// TIA Portal V17 program export: 9 tag tables, 18 data types, 15 data blocks, 39 code blocks (in call order from the OBs), 98 instance data blocks

VAR_GLOBAL   // PLC tag table "Check Scale Station-6"
   TAG_201 AT %M2.3 : Bool;
   TAG_202 AT %M2.4 : Bool;
   Tag_100 AT %M2.5 : Bool;
   "anti jammer_L2" AT %M2.6 : Bool;
   Tag_79_L2 AT %M2.7 : Bool;
   S5_STOPPER_SENSOR_l2 AT %M3.0 : Bool;
   S5_SENSOR_CYL7_DUMMY_TAG AT %M3.1 : Bool;
   Tag_102 AT %M3.2 : Bool;
   Seq_Lifttable_done_L2 AT %M3.3 : Bool;
   MC_Reset_L2 AT %M3.4 : Bool;
   TAG_203 AT %M3.5 : Bool;
   TAG_204 AT %M3.6 : Bool;
   TAG_205 AT %M3.7 : Bool;
   TAG_206 AT %M4.0 : Bool;
   TAG_207 AT %M4.1 : Bool;
   TAG_208 AT %M4.2 : Bool;
   TAG_209 AT %M4.3 : Bool;
   TAG210 AT %M4.4 : Bool;
   TAG211 AT %M4.5 : Bool;
   TAG216 AT %M4.6 : Bool;
   TAG213 AT %M4.7 : Bool;
   TAG214 AT %M5.0 : Bool;
   TAG215 AT %M5.1 : Bool;
   TAG217 AT %M5.2 : Bool;
   TAG218 AT %M5.3 : Bool;
   TAG212 AT %M5.4 : Bool;
   old_id AT %MW6 : Int;
   New_id AT %MW18 : Int;
END_VAR

VAR_GLOBAL   // PLC tag table "Common Tags"
END_VAR

VAR_GLOBAL   // PLC tag table "Correction Station-7"
END_VAR

VAR_GLOBAL   // PLC tag table "Default tag table"
   A_Tag_1 AT %M102.0 : Bool;
   A_Tag_2 AT %M102.1 : Bool;
   A_Tag_3 AT %M102.2 : Bool;
   A_Tag_4 AT %M102.3 : Bool;
   A_Tag_5 AT %M102.4 : Bool;
   Tag_1 AT %M200.0 : Bool;
   P_Trig08 AT %M2.0 : Bool;
   Tag_3 AT %M9.0 : Bool;
   Tag_4 AT %M9.1 : Bool;
   Tag_5 AT %M200.2 : Bool;
   A_Tag_11 AT %M2.1 : Bool;
   Tag_6 AT %M200.1 : Bool;
   Tag_7 AT %M110.0 : Bool;
   Tag_8 AT %M210.0 : Bool;
   Tag_9 AT %M210.1 : Bool;
   Tag_10 AT %M210.2 : Bool;
   Tag_11 AT %M210.4 : Bool;
   Tag_12 AT %M210.5 : Bool;
   Tag_13 AT %M210.6 : Bool;
   temp AT %M300.0 : Bool;
   Tag_14 AT %M210.7 : Bool;
   Tag_15 AT %M9.2 : Bool;
   Tag_17 AT %MW13 : Int;
   Tag_18 AT %MW15 : Int;
   Master1_Done_Bit AT %M11.0 : Bool;
   Master_Error_Bit AT %M11.1 : Bool;
   Tag_19 AT %MW500 : Word;
   Tag_20 AT %MW100 : Int;
   Tag_21 AT %M9.7 : Bool;
   Tag_22 AT %M20.0 : Bool;
   Tag_23 AT %M20.1 : Bool;
   Tag_24 AT %M22.0 : Bool;
   Tag_25 AT %M22.1 : Bool;
   System_Byte AT %MB1 : Byte;
   FirstScan AT %M1.0 : Bool;
   DiagStatusUpdate AT %M1.1 : Bool;
   AlwaysTRUE AT %M1.2 : Bool;
   AlwaysFALSE AT %M1.3 : Bool;
   Clock_Byte AT %MB0 : Byte;
   Clock_10Hz AT %M0.0 : Bool;
   Clock_5Hz AT %M0.1 : Bool;
   "Clock_2.5Hz" AT %M0.2 : Bool;
   Clock_2Hz AT %M0.3 : Bool;
   "Clock_1.25Hz" AT %M0.4 : Bool;
   Clock_1Hz AT %M0.5 : Bool;
   "Clock_0.625Hz" AT %M0.6 : Bool;
   "Clock_0.5Hz" AT %M0.7 : Bool;
   Tag_26 AT %M503.6 : Bool;
   Tag_27 AT %M23.0 : Bool;
   Tag_28 AT %M25.0 : Bool;
   Tag_29 AT %M25.1 : Bool;
   Tag_30 AT %M26.0 : Bool;
   Tag_31 AT %M27.0 : Bool;
   Tag_32 AT %M27.1 : Bool;
   Tag_33 AT %M27.2 : Bool;
   Tag_34 AT %M27.3 : Bool;
   Tag_35 AT %M27.4 : Bool;
   Tag_36 AT %M27.5 : Bool;
   Tag_37 AT %M27.6 : Bool;
   Tag_38 AT %M27.7 : Bool;
   Tag_39 AT %M28.0 : Bool;
   Tag_40 AT %M28.1 : Bool;
   Tag_41 AT %M28.2 : Bool;
   Tag_42 AT %M28.3 : Bool;
   Tag_43 AT %M28.4 : Bool;
   Tag_44 AT %M28.5 : Bool;
   Tag_45 AT %M28.6 : Bool;
   Tag_2 AT %M211.0 : Bool;
   Tag_16 AT %M211.2 : Bool;
   Tag_46 AT %M211.3 : Bool;
   Tag_47 AT %M212.0 : Bool;
   Tag_48 AT %M212.1 : Bool;
   Tag_49 AT %M212.2 : Bool;
   Tag_50 AT %M212.3 : Bool;
   Tag_51 AT %M212.4 : Bool;
   Tag_52 AT %M213.5 : Bool;
   Tag_53 AT %M212.5 : Bool;
   Tag_54 AT %M212.6 : Bool;
   Tag_55 AT %M212.7 : Bool;
   Tag_56 AT %M213.4 : Bool;
   Tag_57 AT %M213.0 : Bool;
   Tag_58 AT %M213.1 : Bool;
   Tag_59 AT %M213.2 : Bool;
   Tag_60 AT %M213.3 : Bool;
   Tag_61 AT %M214.0 : Bool;
   Tag_62 AT %M214.1 : Bool;
   Tag_63 AT %M214.2 : Bool;
   Tag_64 AT %M214.3 : Bool;
   Tag_65 AT %M214.4 : Bool;
   Tag_66 AT %M214.5 : Bool;
   Tag_67 AT %M214.6 : Bool;
   Tag_68 AT %MW1000 : Int;
   Tag_69 AT %M9.3 : Bool;
   Tag_70 AT %M214.7 : Bool;
   NUM_0 AT %I4.0 : Bool;
   NUM_1 AT %I4.1 : Bool;
   NUM_2 AT %I4.2 : Bool;
   NUM_3 AT %I4.3 : Bool;
   NUM_4 AT %I4.4 : Bool;
   NUM_5 AT %I4.5 : Bool;
   NUM_6 AT %I4.6 : Bool;
   NUM_7 AT %I4.7 : Bool;
   NUM_8 AT %I5.0 : Bool;
   NUM_9 AT %I5.1 : Bool;
   ENTER AT %I5.2 : Bool;
   Clear AT %I5.3 : Bool;
   Tag_71 AT %M2.2 : Bool;
   S5_SENSOR_CYL6 AT %I3.6 : Bool;
   S5_DOWN_CONVEYOR AT %I3.7 : Bool;
   SCREEN AT %I5.4 : Bool;
   BPCL_CY AT %I5.5 : Bool;
   MALABAR_GAS AT %I5.6 : Bool;
   "i5.7" AT %I5.7 : Bool;
   "q3.5" AT %Q3.5 : Bool;
   "q3.6" AT %Q3.6 : Bool;
   "q3.7" AT %Q3.7 : Bool;
   Tag_72 AT %M201.0 : Bool;
   Tag_73 AT %M201.1 : Bool;
   Tag_74 AT %M201.2 : Bool;
   Tag_75 AT %M99.7 : Bool;
   cylinder_pos AT %I2.4 : Bool;
   commercial AT %I2.5 : Bool;
   cylinder_exit AT %I2.6 : Bool;
   S5_CYCLE_START_L2 AT %I0.2 : Bool;
   S5_CYCLE_RESET_L2 AT %I0.3 : Bool;
   SEQ_RESET AT %I0.4 : Bool;
   MANUAL_SEQ AT %I0.5 : Bool;
   "i0.6" AT %I0.6 : Bool;
   "i0.7" AT %I0.7 : Bool;
   SEQ_RESET_L2 AT %I2.7 : Bool;
   S5_STOPPER_SENSOR AT %I3.0 : Bool;
   S5_SENSOR_CYL1 AT %I3.1 : Bool;
   S5_SENSOR_CYL2 AT %I3.2 : Bool;
   S5_SENSOR_CYL3 AT %I3.3 : Bool;
   S5_SENSOR_CYL4 AT %I3.4 : Bool;
   S5_SENSOR_CYL5 AT %I3.5 : Bool;
   DIVERTER AT %Q1.4 : Bool;
   PLC_LIVE AT %Q1.5 : Bool;
   spare_2 AT %Q1.6 : Bool;
   spare_3 AT %Q1.7 : Bool;
   S5_STOPPER_OP AT %Q2.0 : Bool;
   S5_LIFT_CYL6 AT %Q2.1 : Bool;
   S5_LIFT_CYL5 AT %Q2.2 : Bool;
   stopper AT %Q0.0 : Bool;
   Tag_76 AT %M888.7 : Bool;
   Tag_77 AT %M888.5 : Bool;
   Tag_78 AT %M888.6 : Bool;
   Seq_Lifttable_done AT %M100.7 : Bool;
   entry_data AT %MW90 : Int;
   MC_Reset AT %M100.2 : Bool;
   Tag_79 AT %M100.4 : Bool;
   "anti jammer" AT %M100.5 : Bool;
   Tag_80 AT %M100.6 : Bool;
   Tag_81 AT %M202.0 : Bool;
   Tag_82 AT %M202.1 : Bool;
   Tag_83 AT %M202.2 : Bool;
   Tag_84 AT %M202.4 : Bool;
   Tag_85 AT %M202.5 : Bool;
   Tag_86 AT %M202.6 : Bool;
   Tag_87 AT %M202.7 : Bool;
   Tag_88 AT %M203.0 : Bool;
   Tag_89 AT %M203.2 : Bool;
   Tag_90 AT %M203.1 : Bool;
   Tag_91 AT %M203.5 : Bool;
   Tag_92 AT %M203.7 : Bool;
   Tag_93 AT %M204.0 : Bool;
   Tag_94 AT %M204.1 : Bool;
   Tag_95 AT %M204.2 : Bool;
   Tag_96 AT %M204.3 : Bool;
   Tag_97 AT %M204.6 : Bool;
   Tag_98 AT %M203.4 : Bool;
   Tag_99 AT %M999.7 : Bool;
   Tag_101 AT %M5.7 : Bool;
   Tag_103 AT %M5.6 : Bool;
   Tag_104 AT %M500.0 : Bool;
   Tag_105 AT %M700.0 : Bool;
   Tag_106 AT %M700.1 : Bool;
   Check_Stopper AT %I6.0 : Bool;
   Check_presence AT %I6.1 : Bool;
   Check_pusher AT %I6.2 : Bool;
   Check_antijammer AT %I6.3 : Bool;
   Check_start_PB AT %I6.4 : Bool;
   Check_reset_PB AT %I6.5 : Bool;
   Check_Down_line_jammer AT %I6.6 : Bool;
   Correction_Stopper_sensor AT %I6.7 : Bool;
   Correction_Lift_sensor AT %I7.0 : Bool;
   Correction_Jammer_sensor AT %I7.1 : Bool;
   Correction_Start_PB AT %I7.2 : Bool;
   Correction_Reset_PB AT %I7.3 : Bool;
   Check_stopper_op AT %Q4.0 : Bool;
   Check_lift_table AT %Q4.1 : Bool;
   Check_pusher_op AT %Q4.2 : Bool;
   Correction_Stopper_solenoid AT %Q4.3 : Bool;
   Correction_Lift_solenoid AT %Q4.4 : Bool;
END_VAR

VAR_GLOBAL   // PLC tag table "Fine Filling Station-4"
   S4_CYCLE_START AT %I0.0 : Bool;
   S4_CYCLE_RESET AT %I0.1 : Bool;
   S4_STOPPER_SENSOR AT %I2.3 : Bool;
   S4_SENSOR_CYL1 AT %I1.1 : Bool;
   S4_SENSOR_CYL2 AT %I1.2 : Bool;
   S4_SENSOR_CYL3 AT %I1.3 : Bool;
   S4_SENSOR_CYL4 AT %I1.4 : Bool;
   S4_SENSOR_CYL5 AT %I1.5 : Bool;
   S4_SENSOR_CYL6 AT %I1.6 : Bool;
   SPARE_1 AT %I1.7 : Bool;
   MANUAL_SEQ_L2 AT %I2.0 : Bool;
   "i0.6_L2" AT %I2.1 : Bool;
   "i0.7_L2" AT %I2.2 : Bool;
   S4_DOWN_CONVEYOR AT %I1.0 : Bool;
   S4_STOPPER_OP AT %Q0.1 : Bool;
   S4_LIFT_CYL1 AT %Q0.2 : Bool;
   S4_LIFT_CYL2 AT %Q0.3 : Bool;
   S4_LIFT_CYL3 AT %Q0.4 : Bool;
   S4_LIFT_CYL4 AT %Q0.5 : Bool;
   S4_LIFT_CYL5 AT %Q0.6 : Bool;
   S4_LIFT_CYL6 AT %Q0.7 : Bool;
   S4_LIFT_CYL7 AT %Q1.0 : Bool;
   S4_LIFT_CYL8 AT %Q1.1 : Bool;
   S4_LIFT_CYL9 AT %Q1.2 : Bool;
   S4_LIFT_CYL10 AT %Q1.3 : Bool;
   S5_LIFT_CYL4 AT %Q2.3 : Bool;
   S5_LIFT_CYL3 AT %Q2.4 : Bool;
   S5_LIFT_CYL2 AT %Q2.5 : Bool;
   S5_LIFT_CYL1 AT %Q2.6 : Bool;
   spare_11 AT %Q2.7 : Bool;
   spare_12 AT %Q3.0 : Bool;
   spare_13 AT %Q3.1 : Bool;
   spare_14 AT %Q3.2 : Bool;
   spare_15 AT %Q3.3 : Bool;
   spare_16 AT %Q3.4 : Bool;
END_VAR

VAR_GLOBAL   // PLC tag table "Fine Filling Station-5"
END_VAR

VAR_GLOBAL   // PLC tag table "Pre Filling Station-2"
END_VAR

VAR_GLOBAL   // PLC tag table "Pre Filling Station-3"
END_VAR

VAR_GLOBAL   // PLC tag table "Tare Entry Station-1"
END_VAR

TYPE "Master_Step_No"
// stored: IsFailsafeCompliant false
   STRUCT
      Master_Step_No : Array[1..6] of USInt;
   END_STRUCT;
END_TYPE

TYPE "Mod_Client_Data"
// stored: IsFailsafeCompliant false
   STRUCT
      request : Bool;
      enable : Bool;
      disconnect : Bool;
      done : Bool;
      busy : Bool;
      error : Bool;
      status : Word;
      statusSave : Word;
      modbusMode : USInt;
      modbusDataAddress : UDInt;
      modbusDataLen : UInt;
   END_STRUCT;
END_TYPE

TYPE "Mod_Connect_Data"
// stored: IsFailsafeCompliant false
   STRUCT
      connectParamClient { S7_SetPoint := 'True'} : TCON_IP_v4;
   END_STRUCT;
   // connectParamClient.InterfaceId := 64;
   // connectParamClient.ID := 16#2;
   // connectParamClient.ActiveEstablished := true;
   // connectParamClient.RemoteAddress.ADDR[1] := 192;
   // connectParamClient.RemoteAddress.ADDR[2] := 168;
   // connectParamClient.RemoteAddress.ADDR[3] := 0;
   // connectParamClient.RemoteAddress.ADDR[4] := 3;
   // connectParamClient.RemotePort := 503;
   // connectParamClient.LocalPort := 0;
END_TYPE

TYPE "Mod_TCP_Data"
// stored: IsFailsafeCompliant false
   STRUCT
      Mod_TCP_Connect : "Mod_Connect_Data";
      Mod_Client { S7_SetPoint := 'True'} : Array[1..6] of "Mod_Client_Data";
   END_STRUCT;
END_TYPE

TYPE "uCylinderData"
// stored: IsFailsafeCompliant false
   STRUCT
      rCylinderID : Int;
      rNet_weight : Real;
      rTareWeight : Real;
      rGross_Weight : Real;
      iCylinderType : Int;   // 0=Domestic Cylinder; 1= Commercial
      iResult : Int;
   END_STRUCT;
END_TYPE

TYPE "ufinefill_station"
// stored: IsFailsafeCompliant false
   STRUCT
      INxNear_Filter_Stopper_L1 : Bool;
      INxFilling_Unit_L2 : Bool;
      INxFilling_Unit_L3 : Bool;
      INxFilling_Unit_L4 : Bool;
      INxFilling_Unit_L5 : Bool;
      INxDown_Line_Conveyor_L6 : Bool;
      INxCylinder_Selection_2 : Bool;
      INxCylinder_Selection_3 : Bool;
      INxCylinder_Selection_4 : Bool;
      INxStopper_Bypass_L2 : Bool;
      INxStopper_Bypass_L3 : Bool;
      INxStopper_Bypass_L4 : Bool;
      OUTxSolenoid_Control_Stopper_L1 : Bool;
      OUTxSolenoid_Control_LiftTable_L2 : Bool;
      OUTxSolenoid_Control_LiftTable_L3 : Bool;
      OUTxSolenoid_Control_LiftTable_L4 : Bool;
      OUTxSolenoid_Control_LiftTable_L5 : Bool;
      iSensingTime : Time;
      OUTxCylinder_Indicator_2 : Bool;
      OUTxCylinder_Indicator_3 : Bool;
      OUTxCylinder_Indicator_4 : Bool;
   END_STRUCT;
END_TYPE

TYPE "ufinefillingstation_general"
// stored: IsFailsafeCompliant false
   STRUCT
      INxCycle_Start : Bool;
      INxCycle_Reset : Bool;
   END_STRUCT;
END_TYPE

TYPE "LPG_CHECK_DATA"
// stored: IsFailsafeCompliant false
   STRUCT
      CHECK_SEQ_IN : Struct
         Cyl_IN_Pos : Bool;
         Auto_Start_Seq : Bool;
         Man_Start_Seq : Bool;
         Stop_Seq : Bool;
         Start_Timeout_Sec : DInt;
         Reset_Seq : Bool;
         Cylinder_Type : Int;
         Tare_Entry_SP : Real;
      END_STRUCT;
      CHECK_SEQ_OUT : Struct
         Checked_Status : Array[1..3] of Bool;
         Domestic_Cyl : Bool;
         Commercial_Cyl : Bool;
         Start_Timeout : Bool;
         Tare_Entry_Error : Bool;
         Filling_Error : Bool;
         Step_No : Int;
         Modbus_Busy : Bool;
      END_STRUCT;
   END_STRUCT;
END_TYPE

TYPE "LPG_FILL_DATA"
// stored: IsFailsafeCompliant false
   STRUCT
      FILL_SEQ_IN : Struct
         Cyl_IN_Pos : Bool;
         Auto_Start_Seq : Bool;
         Man_Start_Seq : Bool;
         Stop_Seq : Bool;
         Start_Timeout_Sec : DInt;
         Reset_Seq : Bool;
         Cylinder_Type : Int;
         Tare_Entry_SP : Real;
      END_STRUCT;
      FILL_SEQ_OUT : Struct
         Filled_Dat : Array[1..3] of Real;
         Domestic_Cyl : Bool;
         Commercial_Cyl : Bool;
         Start_Timeout : Bool;
         Tare_Entry_Error : Bool;
         Filling_Error : Bool;
         Step_No : Int;
         Modbus_Busy : Bool;
      END_STRUCT;
   END_STRUCT;
END_TYPE

TYPE "LPG_FILL_DATA_1"
// stored: IsFailsafeCompliant false
   STRUCT
      FILL_SEQ_IN : Struct
         Cyl_IN_Pos : Bool;
         Auto_Start_Seq : Bool;
         Man_Start_Seq : Bool;
         Stop_Seq : Bool;
         Start_Timeout_Sec : DInt;
         Reset_Seq : Bool;
         Cylinder_Type : Int;
         Tare_Entry_SP : Real;
      END_STRUCT;
      FILL_SEQ_OUT : Struct
         Filled_Dat : Array[1..10] of Real;
         Domestic_Cyl : Bool;
         Commercial_Cyl : Bool;
         Start_Timeout : Bool;
         Tare_Entry_Error : Bool;
         Filling_Error : Bool;
         Step_No : Int;
         Modbus_Busy : Bool;
      END_STRUCT;
   END_STRUCT;
END_TYPE

TYPE "MASTER_STATION"
// stored: IsFailsafeCompliant false
   STRUCT
      MODBUS_MASTER : Array[1..6] of "MOD_MASTER";
   END_STRUCT;
END_TYPE

TYPE "MODBUS_READ"
// stored: IsFailsafeCompliant false
   STRUCT
      MOD_COIL_DATA : Array[1..32] of Bool;
      MOD_HOLD_DATA_1 : Array[1..6] of Word;
      MOD_HOLD_DATA_2 : Array[1..2] of Word;
   END_STRUCT;
   // // MOD_COIL_DATA[1] : Satble Flag
   // // MOD_COIL_DATA[2] : Net Gross Flag
   // // MOD_COIL_DATA[3] : Operating Mode
   // // MOD_COIL_DATA[4] : Start Key Status
   // // MOD_COIL_DATA[5] : Zero Key Status
   // // MOD_COIL_DATA[6] : Tare Key Status
   // // MOD_COIL_DATA[7] : Print Key Status
   // // MOD_COIL_DATA[8] : Power On Zero
   // // MOD_COIL_DATA[9] : One Touch Zero Calibration
   // // MOD_COIL_DATA[10] : Under Weight Flag
   // // MOD_COIL_DATA[11] : Over Weight Flag
   // // MOD_COIL_DATA[12] : Gross Sign
   // // MOD_COIL_DATA[13] : Net Sign
   // // MOD_COIL_DATA[14] : Filled or Checked Data Status(W)
   // // MOD_COIL_DATA[15] : NA
   // // MOD_COIL_DATA[16] : Gate Input
   // // MOD_COIL_DATA[17] : Coarse Output
   // // MOD_COIL_DATA[18] : Fine Output
   // // MOD_COIL_DATA[19] : Batch Over Output
   // // MOD_COIL_DATA[20] : Gate Output
   // // MOD_COIL_DATA[21] : Lifter Output
   // // MOD_COIL_DATA[22] : Jam Output
   // // MOD_COIL_DATA[23] : NA
   // // MOD_COIL_DATA[24] : Indicator is in Parameter / Tare Entry Settings
   // // MOD_COIL_DATA[25] : Filling ON Status
   // // MOD_COIL_DATA[26] : Filling Time Over (W)
   // // MOD_COIL_DATA[27] : Tare Request Status
   // // MOD_COIL_DATA[28] : Filling Over Status
   // // MOD_COIL_DATA[29] : Filling Error Status(W)
   // // MOD_COIL_DATA[30] : Stop Filling (W)
   // // MOD_COIL_DATA[31] : Start Filling (W)
   // // MOD_COIL_DATA[32] : Tare Entry Error
   // // MOD_HOLD_DATA_1[2] : Fiiled Gross Weight
   // // MOD_HOLD_DATA_1[4] : Filled Net Weight
   // // MOD_HOLD_DATA_1[6] : Punched Tare Weight
   // // MOD_HOLD_DATA_2[2] : Fiiled Gross Weight
END_TYPE

TYPE "MODBUS_READ_1"
// stored: IsFailsafeCompliant false
   STRUCT
      MOD_COIL_DATA : Array[1..32] of Bool;
      MOD_HOLD_DATA_1 : Array[1..10] of Word;
      MOD_HOLD_DATA_2 : Array[1..2] of Word;
   END_STRUCT;
   // // MOD_COIL_DATA[1] : Satble Flag
   // // MOD_COIL_DATA[2] : Net Gross Flag
   // // MOD_COIL_DATA[3] : Operating Mode
   // // MOD_COIL_DATA[4] : Start Key Status
   // // MOD_COIL_DATA[5] : Zero Key Status
   // // MOD_COIL_DATA[6] : Tare Key Status
   // // MOD_COIL_DATA[7] : Print Key Status
   // // MOD_COIL_DATA[8] : Power On Zero
   // // MOD_COIL_DATA[9] : One Touch Zero Calibration
   // // MOD_COIL_DATA[10] : Under Weight Flag
   // // MOD_COIL_DATA[11] : Over Weight Flag
   // // MOD_COIL_DATA[12] : Gross Sign
   // // MOD_COIL_DATA[13] : Net Sign
   // // MOD_COIL_DATA[14] : Filled or Checked Data Status(W)
   // // MOD_COIL_DATA[15] : NA
   // // MOD_COIL_DATA[16] : Gate Input
   // // MOD_COIL_DATA[17] : Coarse Output
   // // MOD_COIL_DATA[18] : Fine Output
   // // MOD_COIL_DATA[19] : Batch Over Output
   // // MOD_COIL_DATA[20] : Gate Output
   // // MOD_COIL_DATA[21] : Lifter Output
   // // MOD_COIL_DATA[22] : Jam Output
   // // MOD_COIL_DATA[23] : NA
   // // MOD_COIL_DATA[24] : Indicator is in Parameter / Tare Entry Settings
   // // MOD_COIL_DATA[25] : Filling ON Status
   // // MOD_COIL_DATA[26] : Filling Time Over (W)
   // // MOD_COIL_DATA[27] : Tare Request Status
   // // MOD_COIL_DATA[28] : Filling Over Status
   // // MOD_COIL_DATA[29] : Filling Error Status(W)
   // // MOD_COIL_DATA[30] : Stop Filling (W)
   // // MOD_COIL_DATA[31] : Start Filling (W)
   // // MOD_COIL_DATA[32] : Tare Entry Error
   // // MOD_HOLD_DATA_1[2] : Fiiled Gross Weight
   // // MOD_HOLD_DATA_1[4] : Filled Net Weight
   // // MOD_HOLD_DATA_1[6] : Punched Tare Weight
   // // MOD_HOLD_DATA_2[2] : Fiiled Gross Weight
END_TYPE

TYPE "MODBUS_WRITE"
// stored: IsFailsafeCompliant false
   STRUCT
      MOD_COIL_DATA : Array[1..32] of Bool;
      MOD_HOLD_DATA_1 : Array[1..2] of Word;
      MOD_HOLD_DATA_2 : Array[1..2] of Word;
   END_STRUCT;
   // // MOD_COIL_DATA[1] : Satble Flag
   // // MOD_COIL_DATA[2] : Net Gross Flag
   // // MOD_COIL_DATA[3] : Operating Mode
   // // MOD_COIL_DATA[4] : Start Key Status
   // // MOD_COIL_DATA[5] : Zero Key Status
   // // MOD_COIL_DATA[6] : Tare Key Status
   // // MOD_COIL_DATA[7] : Print Key Status
   // // MOD_COIL_DATA[8] : Power On Zero
   // // MOD_COIL_DATA[9] : One Touch Zero Calibration
   // // MOD_COIL_DATA[10] : Under Weight Flag
   // // MOD_COIL_DATA[11] : Over Weight Flag
   // // MOD_COIL_DATA[12] : Gross Sign
   // // MOD_COIL_DATA[13] : Net Sign
   // // MOD_COIL_DATA[14] : Filled or Checked Data Status(W)
   // // MOD_COIL_DATA[15] : NA
   // // MOD_COIL_DATA[16] : Gate Input
   // // MOD_COIL_DATA[17] : Coarse Output
   // // MOD_COIL_DATA[18] : Fine Output
   // // MOD_COIL_DATA[19] : Batch Over Output
   // // MOD_COIL_DATA[20] : Gate Output
   // // MOD_COIL_DATA[21] : Lifter Output
   // // MOD_COIL_DATA[22] : Jam Output
   // // MOD_COIL_DATA[23] : NA
   // // MOD_COIL_DATA[24] : Indicator is in Parameter / Tare Entry Settings
   // // MOD_COIL_DATA[25] : Filling ON Status
   // // MOD_COIL_DATA[26] : Filling Time Over (W)
   // // MOD_COIL_DATA[27] : Tare Request Status
   // // MOD_COIL_DATA[28] : Filling Over Status
   // // MOD_COIL_DATA[29] : Filling Error Status(W)
   // // MOD_COIL_DATA[30] : Stop Filling (W)
   // // MOD_COIL_DATA[31] : Start Filling (W)
   // // MOD_COIL_DATA[32] : Tare Entry Error
   // // MOD_HOLD_DATA_1[2] : Cylinder Tare Weight
   // // MOD_HOLD_DATA_2[2] : Cylinder Tare Weight
END_TYPE

TYPE "MOD_COMM_LOAD"
// stored: IsFailsafeCompliant false
   STRUCT
      BAUD : UDInt;
      PARITY : UInt;
      FLOW_CTRL : UInt;
      RTS_ON_DLY : UInt;
      RTS_OFF_DLY : UInt;
      RESP_TO : UInt;
      DONE : Bool;
      ERROR : Bool;
      STATUS : Word;
   END_STRUCT;
END_TYPE

TYPE "MOD_MASTER"
// stored: IsFailsafeCompliant false
   STRUCT
      REQ : Bool;
      ADDR : UInt;
      MODE : USInt;
      DATA_ADDR : UDInt;
      DATA_LEN : UInt;
      DONE : Bool;
      BUSY : Bool;
      ERROR : Bool;
      STATUS : Word;
   END_STRUCT;
END_TYPE

TYPE "MOD_MASTER_DATA"
// stored: IsFailsafeCompliant false
   STRUCT
      MASTER_READ_DATA { S7_SetPoint := 'True'} : "MODBUS_READ";
      MASTER_WRITE_DATA { S7_SetPoint := 'True'} : "MODBUS_WRITE";
   END_STRUCT;
END_TYPE

TYPE "MOD_MASTER_DATA_1"
// stored: IsFailsafeCompliant false
   STRUCT
      MASTER_READ_DATA { S7_SetPoint := 'True'} : "MODBUS_READ_1";
      MASTER_WRITE_DATA { S7_SetPoint := 'True'} : "MODBUS_WRITE";
   END_STRUCT;
END_TYPE

DATA_BLOCK "Check_scale_Report"   // DB2001
{ S7_Optimized_Access := 'TRUE' }
VERSION : 0.1
// stored: AutoNumber false, DBAccessibleFromOPCUA true, IsOnlyStoredInLoadMemory false, IsRetainMemResEnabled false, IsWriteProtectedInAS false, MemoryReserve 100
   VAR
      Check_SCALE_DATA : "uCylinderData";
      Check_SCALE_DONE { S7_SetPoint := 'True'} : Bool;
   END_VAR
BEGIN
END_DATA_BLOCK

DATA_BLOCK "MASTER_FILL_DATA"   // DB105
{ S7_Optimized_Access := 'FALSE' }
VERSION : 0.1
// stored: AutoNumber false, DBAccessibleFromOPCUA true, IsOnlyStoredInLoadMemory false, IsWriteProtectedInAS false
   VAR
      FILL_STATION_4 : Array[1..6] of "LPG_FILL_DATA";
      FILL_STATION_5 : Array[1..6] of "LPG_FILL_DATA";
      CHECK_SCALE_1 { S7_SetPoint := 'True'} : "LPG_FILL_DATA_1";
      CORRECTION_SCALE { S7_SetPoint := 'True'} : "LPG_FILL_DATA";
   END_VAR
BEGIN
END_DATA_BLOCK

DATA_BLOCK "MASTER_SETUP_DB"   // DB13
{ S7_Optimized_Access := 'FALSE' }
VERSION : 0.1
// stored: AutoNumber true, DBAccessibleFromOPCUA true, IsOnlyStoredInLoadMemory false, IsWriteProtectedInAS false
   VAR RETAIN
      Enable_Station1 : Bool;
      Enable_Station4 : Bool;
      S1_Enabled_Station : Array[1..6] of Bool;
      S4_Enabled_Station : Array[1..6] of Bool;
      S1_Total_Station : Int;
      S4_Total_Station : Int;
      Enabled_Station_S1 : Int;
      Enabled_Station_S4 : Int;
      Enabled_Station_S5 : Int;
      S5_Enabled_Station : Array[1..6] of Bool;
      S5_Total_Station : Int;
      Enable_Station5 : Bool;
   END_VAR
BEGIN
END_DATA_BLOCK

DATA_BLOCK "MASTER_TCP_DATA"   // DB104
{ S7_Optimized_Access := 'FALSE' }
VERSION : 0.1
// stored: AutoNumber false, DBAccessibleFromOPCUA true, IsOnlyStoredInLoadMemory false, IsWriteProtectedInAS false
   VAR
      MOD_DEVICE_STATION4 : Array[1..6] of "MOD_MASTER_DATA";
      MOD_DEVICE_STATION5 : Array[1..6] of "MOD_MASTER_DATA";
      CHECK_SCALE_1 { S7_SetPoint := 'True'} : "MOD_MASTER_DATA_1";
      CORRECTION_SCALE { S7_SetPoint := 'True'} : "MOD_MASTER_DATA_1";
   END_VAR
BEGIN
END_DATA_BLOCK

DATA_BLOCK "MODBUS_DATA_READ"   // DB101
{ S7_Optimized_Access := 'FALSE' }
VERSION : 0.1
// stored: AutoNumber false, DBAccessibleFromOPCUA true, IsOnlyStoredInLoadMemory false, IsWriteProtectedInAS false
   VAR
      MOD_RD_DEV_STN4 : Array[1..6] of "MODBUS_READ";
      MOD_RD_DEV_STN5 : Array[1..6] of "MODBUS_READ";
      MOD_RD_DEV_CHECK_SCALE { S7_SetPoint := 'True'} : "MODBUS_READ_1";
      MOD_RD_DEV_CORRECTION_SCALE { S7_SetPoint := 'True'} : "MODBUS_READ_1";
   END_VAR
BEGIN
END_DATA_BLOCK

DATA_BLOCK "MODBUS_DATA_WRITE"   // DB102
{ S7_Optimized_Access := 'FALSE' }
VERSION : 0.1
// stored: AutoNumber false, DBAccessibleFromOPCUA true, IsOnlyStoredInLoadMemory false, IsWriteProtectedInAS false
   VAR
      MOD_WR_DEV_STN4 : Array[1..6] of "MODBUS_WRITE";
      MOD_WR_DEV_STN5 : Array[1..6] of "MODBUS_WRITE";
      MOD_WR_DEV_CHECK_SCALE_1 { S7_SetPoint := 'True'} : "MODBUS_WRITE";
      MOD_WR_DEV_CORRECTION_SCALE { S7_SetPoint := 'True'} : "MODBUS_WRITE";
   END_VAR
BEGIN
END_DATA_BLOCK

DATA_BLOCK "MOD_TCP_SETUP_DB"   // DB100
{ S7_Optimized_Access := 'FALSE' }
VERSION : 0.1
// stored: AutoNumber false, DBAccessibleFromOPCUA true, IsOnlyStoredInLoadMemory false, IsWriteProtectedInAS false
   VAR RETAIN
      TCP_Data_Station4 { ExternalAccessible := 'False'; ExternalVisible := 'False'; ExternalWritable := 'False'; S7_SetPoint := 'True'} : Array[1..6] of "Mod_TCP_Data";
      TCP_Data_Station5 { ExternalAccessible := 'False'; ExternalVisible := 'False'; ExternalWritable := 'False'} : Array[1..6] of "Mod_TCP_Data";
      TCP_Data_CHECK_SCALE_1 { S7_SetPoint := 'True'} : "Mod_TCP_Data";
      TCP_Data_CORRECTION_SCALE { S7_SetPoint := 'True'} : "Mod_TCP_Data";
   END_VAR
BEGIN
   TCP_Data_Station4[1..6].Mod_TCP_Connect.connectParamClient.InterfaceId := 64;
   TCP_Data_Station4[1].Mod_TCP_Connect.connectParamClient.ID := 1;
   TCP_Data_Station4[2].Mod_TCP_Connect.connectParamClient.ID := 2;
   TCP_Data_Station4[3].Mod_TCP_Connect.connectParamClient.ID := 3;
   TCP_Data_Station4[4].Mod_TCP_Connect.connectParamClient.ID := 4;
   TCP_Data_Station4[5].Mod_TCP_Connect.connectParamClient.ID := 5;
   TCP_Data_Station4[6].Mod_TCP_Connect.connectParamClient.ID := 6;
   TCP_Data_Station4[1..6].Mod_TCP_Connect.connectParamClient.ConnectionType := 16#0B;
   TCP_Data_Station4[1..6].Mod_TCP_Connect.connectParamClient.ActiveEstablished := true;
   TCP_Data_Station4[1].Mod_TCP_Connect.connectParamClient.RemoteAddress.ADDR[1] := 192;
   TCP_Data_Station4[1].Mod_TCP_Connect.connectParamClient.RemoteAddress.ADDR[2] := 168;
   TCP_Data_Station4[1].Mod_TCP_Connect.connectParamClient.RemoteAddress.ADDR[3] := 0;
   TCP_Data_Station4[1].Mod_TCP_Connect.connectParamClient.RemoteAddress.ADDR[4] := 21;
   TCP_Data_Station4[2].Mod_TCP_Connect.connectParamClient.RemoteAddress.ADDR[1] := 192;
   TCP_Data_Station4[2].Mod_TCP_Connect.connectParamClient.RemoteAddress.ADDR[2] := 168;
   TCP_Data_Station4[2].Mod_TCP_Connect.connectParamClient.RemoteAddress.ADDR[3] := 0;
   TCP_Data_Station4[2].Mod_TCP_Connect.connectParamClient.RemoteAddress.ADDR[4] := 22;
   TCP_Data_Station4[3].Mod_TCP_Connect.connectParamClient.RemoteAddress.ADDR[1] := 192;
   TCP_Data_Station4[3].Mod_TCP_Connect.connectParamClient.RemoteAddress.ADDR[2] := 168;
   TCP_Data_Station4[3].Mod_TCP_Connect.connectParamClient.RemoteAddress.ADDR[3] := 0;
   TCP_Data_Station4[3].Mod_TCP_Connect.connectParamClient.RemoteAddress.ADDR[4] := 23;
   TCP_Data_Station4[4].Mod_TCP_Connect.connectParamClient.RemoteAddress.ADDR[1] := 192;
   TCP_Data_Station4[4].Mod_TCP_Connect.connectParamClient.RemoteAddress.ADDR[2] := 168;
   TCP_Data_Station4[4].Mod_TCP_Connect.connectParamClient.RemoteAddress.ADDR[3] := 0;
   TCP_Data_Station4[4].Mod_TCP_Connect.connectParamClient.RemoteAddress.ADDR[4] := 24;
   TCP_Data_Station4[5].Mod_TCP_Connect.connectParamClient.RemoteAddress.ADDR[1] := 192;
   TCP_Data_Station4[5].Mod_TCP_Connect.connectParamClient.RemoteAddress.ADDR[2] := 168;
   TCP_Data_Station4[5].Mod_TCP_Connect.connectParamClient.RemoteAddress.ADDR[3] := 0;
   TCP_Data_Station4[5].Mod_TCP_Connect.connectParamClient.RemoteAddress.ADDR[4] := 25;
   TCP_Data_Station4[6].Mod_TCP_Connect.connectParamClient.RemoteAddress.ADDR[1] := 192;
   TCP_Data_Station4[6].Mod_TCP_Connect.connectParamClient.RemoteAddress.ADDR[2] := 168;
   TCP_Data_Station4[6].Mod_TCP_Connect.connectParamClient.RemoteAddress.ADDR[3] := 0;
   TCP_Data_Station4[6].Mod_TCP_Connect.connectParamClient.RemoteAddress.ADDR[4] := 26;
   TCP_Data_Station4[1..6].Mod_TCP_Connect.connectParamClient.RemotePort := 502;
   TCP_Data_Station4[2..6].Mod_TCP_Connect.connectParamClient.LocalPort := 0;
   TCP_Data_Station4[1].Mod_Client[1..6].request := false;
   TCP_Data_Station4[2].Mod_Client[1..6].request := false;
   TCP_Data_Station4[3].Mod_Client[1..6].request := false;
   TCP_Data_Station4[4].Mod_Client[1..6].request := false;
   TCP_Data_Station4[5].Mod_Client[1..6].request := false;
   TCP_Data_Station4[6].Mod_Client[1..6].request := false;
   TCP_Data_Station4[1].Mod_Client[1..6].enable := false;
   TCP_Data_Station4[2].Mod_Client[1..6].enable := false;
   TCP_Data_Station4[3].Mod_Client[1..6].enable := false;
   TCP_Data_Station4[4].Mod_Client[1..6].enable := false;
   TCP_Data_Station4[5].Mod_Client[1..6].enable := false;
   TCP_Data_Station4[6].Mod_Client[1..6].enable := false;
   TCP_Data_Station4[1].Mod_Client[1..6].disconnect := false;
   TCP_Data_Station4[2].Mod_Client[1..6].disconnect := false;
   TCP_Data_Station4[3].Mod_Client[1..6].disconnect := false;
   TCP_Data_Station4[4].Mod_Client[1..6].disconnect := false;
   TCP_Data_Station4[5].Mod_Client[1..6].disconnect := false;
   TCP_Data_Station4[6].Mod_Client[1..6].disconnect := false;
   TCP_Data_Station4[1].Mod_Client[1..6].done := false;
   TCP_Data_Station4[2].Mod_Client[1..6].done := false;
   TCP_Data_Station4[3].Mod_Client[1..6].done := false;
   TCP_Data_Station4[4].Mod_Client[1..6].done := false;
   TCP_Data_Station4[5].Mod_Client[1..6].done := false;
   TCP_Data_Station4[6].Mod_Client[1..6].done := false;
   TCP_Data_Station4[1].Mod_Client[1..6].busy := false;
   TCP_Data_Station4[2].Mod_Client[1..6].busy := false;
   TCP_Data_Station4[3].Mod_Client[1..6].busy := false;
   TCP_Data_Station4[4].Mod_Client[1..6].busy := false;
   TCP_Data_Station4[5].Mod_Client[1..6].busy := false;
   TCP_Data_Station4[6].Mod_Client[1..6].busy := false;
   TCP_Data_Station4[1].Mod_Client[1..6].error := false;
   TCP_Data_Station4[2].Mod_Client[1..6].error := false;
   TCP_Data_Station4[3].Mod_Client[1..6].error := false;
   TCP_Data_Station4[4].Mod_Client[1..6].error := false;
   TCP_Data_Station4[5].Mod_Client[1..6].error := false;
   TCP_Data_Station4[6].Mod_Client[1..6].error := false;
   TCP_Data_Station4[1].Mod_Client[1..6].status := 16#0;
   TCP_Data_Station4[2].Mod_Client[1..6].status := 16#0;
   TCP_Data_Station4[3].Mod_Client[1..6].status := 16#0;
   TCP_Data_Station4[4].Mod_Client[1..6].status := 16#0;
   TCP_Data_Station4[5].Mod_Client[1..6].status := 16#0;
   TCP_Data_Station4[6].Mod_Client[1..6].status := 16#0;
   TCP_Data_Station4[1].Mod_Client[1..6].statusSave := 16#0;
   TCP_Data_Station4[2].Mod_Client[1..6].statusSave := 16#0;
   TCP_Data_Station4[3].Mod_Client[1..6].statusSave := 16#0;
   TCP_Data_Station4[4].Mod_Client[1..6].statusSave := 16#0;
   TCP_Data_Station4[5].Mod_Client[1..6].statusSave := 16#0;
   TCP_Data_Station4[6].Mod_Client[1..6].statusSave := 16#0;
   TCP_Data_Station4[1].Mod_Client[1].modbusMode := 1;
   TCP_Data_Station4[1].Mod_Client[2].modbusMode := 0;
   TCP_Data_Station4[1].Mod_Client[3].modbusMode := 1;
   TCP_Data_Station4[1].Mod_Client[4..5].modbusMode := 0;
   TCP_Data_Station4[1].Mod_Client[6].modbusMode := 1;
   TCP_Data_Station4[2].Mod_Client[1].modbusMode := 1;
   TCP_Data_Station4[2].Mod_Client[2].modbusMode := 0;
   TCP_Data_Station4[2].Mod_Client[3].modbusMode := 1;
   TCP_Data_Station4[2].Mod_Client[4..5].modbusMode := 0;
   TCP_Data_Station4[2].Mod_Client[6].modbusMode := 1;
   TCP_Data_Station4[3].Mod_Client[1].modbusMode := 1;
   TCP_Data_Station4[3].Mod_Client[2].modbusMode := 0;
   TCP_Data_Station4[3].Mod_Client[3].modbusMode := 1;
   TCP_Data_Station4[3].Mod_Client[4..5].modbusMode := 0;
   TCP_Data_Station4[3].Mod_Client[6].modbusMode := 1;
   TCP_Data_Station4[4].Mod_Client[1].modbusMode := 1;
   TCP_Data_Station4[4].Mod_Client[2].modbusMode := 0;
   TCP_Data_Station4[4].Mod_Client[3].modbusMode := 1;
   TCP_Data_Station4[4].Mod_Client[4..5].modbusMode := 0;
   TCP_Data_Station4[4].Mod_Client[6].modbusMode := 1;
   TCP_Data_Station4[5].Mod_Client[1].modbusMode := 1;
   TCP_Data_Station4[5].Mod_Client[2].modbusMode := 0;
   TCP_Data_Station4[5].Mod_Client[3].modbusMode := 1;
   TCP_Data_Station4[5].Mod_Client[4..5].modbusMode := 0;
   TCP_Data_Station4[5].Mod_Client[6].modbusMode := 1;
   TCP_Data_Station4[6].Mod_Client[1].modbusMode := 1;
   TCP_Data_Station4[6].Mod_Client[2].modbusMode := 0;
   TCP_Data_Station4[6].Mod_Client[3].modbusMode := 1;
   TCP_Data_Station4[6].Mod_Client[4..5].modbusMode := 0;
   TCP_Data_Station4[6].Mod_Client[6].modbusMode := 1;
   TCP_Data_Station4[1].Mod_Client[1].modbusDataAddress := 40908;
   TCP_Data_Station4[1].Mod_Client[2].modbusDataAddress := 40001;
   TCP_Data_Station4[1].Mod_Client[3].modbusDataAddress := 40302;
   TCP_Data_Station4[1].Mod_Client[4].modbusDataAddress := 0;
   TCP_Data_Station4[1].Mod_Client[5].modbusDataAddress := 1;
   TCP_Data_Station4[1].Mod_Client[6].modbusDataAddress := 0;
   TCP_Data_Station4[2].Mod_Client[1].modbusDataAddress := 40908;
   TCP_Data_Station4[2].Mod_Client[2].modbusDataAddress := 40001;
   TCP_Data_Station4[2].Mod_Client[3].modbusDataAddress := 40302;
   TCP_Data_Station4[2].Mod_Client[4].modbusDataAddress := 0;
   TCP_Data_Station4[2].Mod_Client[5].modbusDataAddress := 1;
   TCP_Data_Station4[2].Mod_Client[6].modbusDataAddress := 0;
   TCP_Data_Station4[3].Mod_Client[1].modbusDataAddress := 40908;
   TCP_Data_Station4[3].Mod_Client[2].modbusDataAddress := 40001;
   TCP_Data_Station4[3].Mod_Client[3].modbusDataAddress := 40302;
   TCP_Data_Station4[3].Mod_Client[4].modbusDataAddress := 0;
   TCP_Data_Station4[3].Mod_Client[5].modbusDataAddress := 1;
   TCP_Data_Station4[3].Mod_Client[6].modbusDataAddress := 0;
   TCP_Data_Station4[4].Mod_Client[1].modbusDataAddress := 40908;
   TCP_Data_Station4[4].Mod_Client[2].modbusDataAddress := 40001;
   TCP_Data_Station4[4].Mod_Client[3].modbusDataAddress := 40302;
   TCP_Data_Station4[4].Mod_Client[4].modbusDataAddress := 0;
   TCP_Data_Station4[4].Mod_Client[5].modbusDataAddress := 1;
   TCP_Data_Station4[4].Mod_Client[6].modbusDataAddress := 0;
   TCP_Data_Station4[5].Mod_Client[1].modbusDataAddress := 40908;
   TCP_Data_Station4[5].Mod_Client[2].modbusDataAddress := 40001;
   TCP_Data_Station4[5].Mod_Client[3].modbusDataAddress := 40302;
   TCP_Data_Station4[5].Mod_Client[4].modbusDataAddress := 0;
   TCP_Data_Station4[5].Mod_Client[5].modbusDataAddress := 1;
   TCP_Data_Station4[5].Mod_Client[6].modbusDataAddress := 0;
   TCP_Data_Station4[6].Mod_Client[1].modbusDataAddress := 40908;
   TCP_Data_Station4[6].Mod_Client[2].modbusDataAddress := 40001;
   TCP_Data_Station4[6].Mod_Client[3].modbusDataAddress := 40302;
   TCP_Data_Station4[6].Mod_Client[4].modbusDataAddress := 0;
   TCP_Data_Station4[6].Mod_Client[5].modbusDataAddress := 1;
   TCP_Data_Station4[6].Mod_Client[6].modbusDataAddress := 0;
   TCP_Data_Station4[1].Mod_Client[1].modbusDataLen := 1;
   TCP_Data_Station4[1].Mod_Client[2].modbusDataLen := 6;
   TCP_Data_Station4[1].Mod_Client[3].modbusDataLen := 1;
   TCP_Data_Station4[1].Mod_Client[4].modbusDataLen := 0;
   TCP_Data_Station4[1].Mod_Client[5].modbusDataLen := 32;
   TCP_Data_Station4[1].Mod_Client[6].modbusDataLen := 1;
   TCP_Data_Station4[2].Mod_Client[1].modbusDataLen := 1;
   TCP_Data_Station4[2].Mod_Client[2].modbusDataLen := 6;
   TCP_Data_Station4[2].Mod_Client[3].modbusDataLen := 1;
   TCP_Data_Station4[2].Mod_Client[4].modbusDataLen := 0;
   TCP_Data_Station4[2].Mod_Client[5].modbusDataLen := 32;
   TCP_Data_Station4[2].Mod_Client[6].modbusDataLen := 1;
   TCP_Data_Station4[3].Mod_Client[1].modbusDataLen := 1;
   TCP_Data_Station4[3].Mod_Client[2].modbusDataLen := 6;
   TCP_Data_Station4[3].Mod_Client[3].modbusDataLen := 1;
   TCP_Data_Station4[3].Mod_Client[4].modbusDataLen := 0;
   TCP_Data_Station4[3].Mod_Client[5].modbusDataLen := 32;
   TCP_Data_Station4[3].Mod_Client[6].modbusDataLen := 1;
   TCP_Data_Station4[4].Mod_Client[1].modbusDataLen := 1;
   TCP_Data_Station4[4].Mod_Client[2].modbusDataLen := 6;
   TCP_Data_Station4[4].Mod_Client[3].modbusDataLen := 1;
   TCP_Data_Station4[4].Mod_Client[4].modbusDataLen := 0;
   TCP_Data_Station4[4].Mod_Client[5].modbusDataLen := 32;
   TCP_Data_Station4[4].Mod_Client[6].modbusDataLen := 1;
   TCP_Data_Station4[5].Mod_Client[1].modbusDataLen := 1;
   TCP_Data_Station4[5].Mod_Client[2].modbusDataLen := 6;
   TCP_Data_Station4[5].Mod_Client[3].modbusDataLen := 1;
   TCP_Data_Station4[5].Mod_Client[4].modbusDataLen := 0;
   TCP_Data_Station4[5].Mod_Client[5].modbusDataLen := 32;
   TCP_Data_Station4[5].Mod_Client[6].modbusDataLen := 1;
   TCP_Data_Station4[6].Mod_Client[1].modbusDataLen := 1;
   TCP_Data_Station4[6].Mod_Client[2].modbusDataLen := 6;
   TCP_Data_Station4[6].Mod_Client[3].modbusDataLen := 1;
   TCP_Data_Station4[6].Mod_Client[4].modbusDataLen := 0;
   TCP_Data_Station4[6].Mod_Client[5].modbusDataLen := 32;
   TCP_Data_Station4[6].Mod_Client[6].modbusDataLen := 1;
   TCP_Data_Station5[1..6].Mod_TCP_Connect.connectParamClient.InterfaceId := 64;
   TCP_Data_Station5[1].Mod_TCP_Connect.connectParamClient.ID := 11;
   TCP_Data_Station5[2].Mod_TCP_Connect.connectParamClient.ID := 12;
   TCP_Data_Station5[3].Mod_TCP_Connect.connectParamClient.ID := 13;
   TCP_Data_Station5[4].Mod_TCP_Connect.connectParamClient.ID := 14;
   TCP_Data_Station5[5].Mod_TCP_Connect.connectParamClient.ID := 15;
   TCP_Data_Station5[6].Mod_TCP_Connect.connectParamClient.ID := 16;
   TCP_Data_Station5[1..6].Mod_TCP_Connect.connectParamClient.ConnectionType := 16#0B;
   TCP_Data_Station5[1].Mod_TCP_Connect.connectParamClient.ActiveEstablished := true;
   TCP_Data_Station5[2..6].Mod_TCP_Connect.connectParamClient.ActiveEstablished := True;
   TCP_Data_Station5[1].Mod_TCP_Connect.connectParamClient.RemoteAddress.ADDR[1] := 192;
   TCP_Data_Station5[1].Mod_TCP_Connect.connectParamClient.RemoteAddress.ADDR[2] := 168;
   TCP_Data_Station5[1].Mod_TCP_Connect.connectParamClient.RemoteAddress.ADDR[3] := 0;
   TCP_Data_Station5[1].Mod_TCP_Connect.connectParamClient.RemoteAddress.ADDR[4] := 31;
   TCP_Data_Station5[2].Mod_TCP_Connect.connectParamClient.RemoteAddress.ADDR[1] := 192;
   TCP_Data_Station5[2].Mod_TCP_Connect.connectParamClient.RemoteAddress.ADDR[2] := 168;
   TCP_Data_Station5[2].Mod_TCP_Connect.connectParamClient.RemoteAddress.ADDR[3] := 0;
   TCP_Data_Station5[2].Mod_TCP_Connect.connectParamClient.RemoteAddress.ADDR[4] := 32;
   TCP_Data_Station5[3].Mod_TCP_Connect.connectParamClient.RemoteAddress.ADDR[1] := 192;
   TCP_Data_Station5[3].Mod_TCP_Connect.connectParamClient.RemoteAddress.ADDR[2] := 168;
   TCP_Data_Station5[3].Mod_TCP_Connect.connectParamClient.RemoteAddress.ADDR[3] := 0;
   TCP_Data_Station5[3].Mod_TCP_Connect.connectParamClient.RemoteAddress.ADDR[4] := 33;
   TCP_Data_Station5[4].Mod_TCP_Connect.connectParamClient.RemoteAddress.ADDR[1] := 192;
   TCP_Data_Station5[4].Mod_TCP_Connect.connectParamClient.RemoteAddress.ADDR[2] := 168;
   TCP_Data_Station5[4].Mod_TCP_Connect.connectParamClient.RemoteAddress.ADDR[3] := 0;
   TCP_Data_Station5[4].Mod_TCP_Connect.connectParamClient.RemoteAddress.ADDR[4] := 34;
   TCP_Data_Station5[5].Mod_TCP_Connect.connectParamClient.RemoteAddress.ADDR[1] := 192;
   TCP_Data_Station5[5].Mod_TCP_Connect.connectParamClient.RemoteAddress.ADDR[2] := 168;
   TCP_Data_Station5[5].Mod_TCP_Connect.connectParamClient.RemoteAddress.ADDR[3] := 0;
   TCP_Data_Station5[5].Mod_TCP_Connect.connectParamClient.RemoteAddress.ADDR[4] := 35;
   TCP_Data_Station5[6].Mod_TCP_Connect.connectParamClient.RemoteAddress.ADDR[1] := 192;
   TCP_Data_Station5[6].Mod_TCP_Connect.connectParamClient.RemoteAddress.ADDR[2] := 168;
   TCP_Data_Station5[6].Mod_TCP_Connect.connectParamClient.RemoteAddress.ADDR[3] := 0;
   TCP_Data_Station5[6].Mod_TCP_Connect.connectParamClient.RemoteAddress.ADDR[4] := 36;
   TCP_Data_Station5[1..6].Mod_TCP_Connect.connectParamClient.RemotePort := 502;
   TCP_Data_Station5[1..6].Mod_TCP_Connect.connectParamClient.LocalPort := 0;
   TCP_Data_Station5[1].Mod_Client[1..6].request := false;
   TCP_Data_Station5[2].Mod_Client[1..6].request := false;
   TCP_Data_Station5[3].Mod_Client[1..6].request := false;
   TCP_Data_Station5[4].Mod_Client[1..6].request := false;
   TCP_Data_Station5[5].Mod_Client[1..6].request := false;
   TCP_Data_Station5[6].Mod_Client[1..6].request := false;
   TCP_Data_Station5[1].Mod_Client[1..6].enable := false;
   TCP_Data_Station5[2].Mod_Client[1..6].enable := false;
   TCP_Data_Station5[3].Mod_Client[1..6].enable := false;
   TCP_Data_Station5[4].Mod_Client[1..6].enable := false;
   TCP_Data_Station5[5].Mod_Client[1..6].enable := false;
   TCP_Data_Station5[6].Mod_Client[1..6].enable := false;
   TCP_Data_Station5[1].Mod_Client[1..6].disconnect := false;
   TCP_Data_Station5[2].Mod_Client[1..6].disconnect := false;
   TCP_Data_Station5[3].Mod_Client[1..6].disconnect := false;
   TCP_Data_Station5[4].Mod_Client[1..6].disconnect := false;
   TCP_Data_Station5[5].Mod_Client[1..6].disconnect := false;
   TCP_Data_Station5[6].Mod_Client[1..6].disconnect := false;
   TCP_Data_Station5[1].Mod_Client[1..6].done := false;
   TCP_Data_Station5[2].Mod_Client[1..6].done := false;
   TCP_Data_Station5[3].Mod_Client[1..6].done := false;
   TCP_Data_Station5[4].Mod_Client[1..6].done := false;
   TCP_Data_Station5[5].Mod_Client[1..6].done := false;
   TCP_Data_Station5[6].Mod_Client[1..6].done := false;
   TCP_Data_Station5[1].Mod_Client[1..6].busy := false;
   TCP_Data_Station5[2].Mod_Client[1..6].busy := false;
   TCP_Data_Station5[3].Mod_Client[1..6].busy := false;
   TCP_Data_Station5[4].Mod_Client[1..6].busy := false;
   TCP_Data_Station5[5].Mod_Client[1..6].busy := false;
   TCP_Data_Station5[6].Mod_Client[1..6].busy := false;
   TCP_Data_Station5[1].Mod_Client[1..6].error := false;
   TCP_Data_Station5[2].Mod_Client[1..6].error := false;
   TCP_Data_Station5[3].Mod_Client[1..6].error := false;
   TCP_Data_Station5[4].Mod_Client[1..6].error := false;
   TCP_Data_Station5[5].Mod_Client[1..6].error := false;
   TCP_Data_Station5[6].Mod_Client[1..6].error := false;
   TCP_Data_Station5[1].Mod_Client[1..6].status := 16#0;
   TCP_Data_Station5[2].Mod_Client[1..6].status := 16#0;
   TCP_Data_Station5[3].Mod_Client[1..6].status := 16#0;
   TCP_Data_Station5[4].Mod_Client[1..6].status := 16#0;
   TCP_Data_Station5[5].Mod_Client[1..6].status := 16#0;
   TCP_Data_Station5[6].Mod_Client[1..6].status := 16#0;
   TCP_Data_Station5[1].Mod_Client[1..6].statusSave := 16#0;
   TCP_Data_Station5[2].Mod_Client[1..6].statusSave := 16#0;
   TCP_Data_Station5[3].Mod_Client[1..6].statusSave := 16#0;
   TCP_Data_Station5[4].Mod_Client[1..6].statusSave := 16#0;
   TCP_Data_Station5[5].Mod_Client[1..6].statusSave := 16#0;
   TCP_Data_Station5[6].Mod_Client[1..6].statusSave := 16#0;
   TCP_Data_Station5[1].Mod_Client[1].modbusMode := 1;
   TCP_Data_Station5[1].Mod_Client[2].modbusMode := 0;
   TCP_Data_Station5[1].Mod_Client[3].modbusMode := 1;
   TCP_Data_Station5[1].Mod_Client[4..5].modbusMode := 0;
   TCP_Data_Station5[1].Mod_Client[6].modbusMode := 1;
   TCP_Data_Station5[2].Mod_Client[1].modbusMode := 1;
   TCP_Data_Station5[2].Mod_Client[2].modbusMode := 0;
   TCP_Data_Station5[2].Mod_Client[3].modbusMode := 1;
   TCP_Data_Station5[2].Mod_Client[4..5].modbusMode := 0;
   TCP_Data_Station5[2].Mod_Client[6].modbusMode := 1;
   TCP_Data_Station5[3].Mod_Client[1].modbusMode := 1;
   TCP_Data_Station5[3].Mod_Client[2].modbusMode := 0;
   TCP_Data_Station5[3].Mod_Client[3].modbusMode := 1;
   TCP_Data_Station5[3].Mod_Client[4..5].modbusMode := 0;
   TCP_Data_Station5[3].Mod_Client[6].modbusMode := 1;
   TCP_Data_Station5[4].Mod_Client[1].modbusMode := 1;
   TCP_Data_Station5[4].Mod_Client[2].modbusMode := 0;
   TCP_Data_Station5[4].Mod_Client[3].modbusMode := 1;
   TCP_Data_Station5[4].Mod_Client[4..5].modbusMode := 0;
   TCP_Data_Station5[4].Mod_Client[6].modbusMode := 1;
   TCP_Data_Station5[5].Mod_Client[1].modbusMode := 1;
   TCP_Data_Station5[5].Mod_Client[2].modbusMode := 0;
   TCP_Data_Station5[5].Mod_Client[3].modbusMode := 1;
   TCP_Data_Station5[5].Mod_Client[4..5].modbusMode := 0;
   TCP_Data_Station5[5].Mod_Client[6].modbusMode := 1;
   TCP_Data_Station5[6].Mod_Client[1].modbusMode := 1;
   TCP_Data_Station5[6].Mod_Client[2].modbusMode := 0;
   TCP_Data_Station5[6].Mod_Client[3].modbusMode := 1;
   TCP_Data_Station5[6].Mod_Client[4..5].modbusMode := 0;
   TCP_Data_Station5[6].Mod_Client[6].modbusMode := 1;
   TCP_Data_Station5[1].Mod_Client[1].modbusDataAddress := 40908;
   TCP_Data_Station5[1].Mod_Client[2].modbusDataAddress := 40001;
   TCP_Data_Station5[1].Mod_Client[3].modbusDataAddress := 40302;
   TCP_Data_Station5[1].Mod_Client[4].modbusDataAddress := 0;
   TCP_Data_Station5[1].Mod_Client[5].modbusDataAddress := 1;
   TCP_Data_Station5[1].Mod_Client[6].modbusDataAddress := 0;
   TCP_Data_Station5[2].Mod_Client[1].modbusDataAddress := 40908;
   TCP_Data_Station5[2].Mod_Client[2].modbusDataAddress := 40001;
   TCP_Data_Station5[2].Mod_Client[3].modbusDataAddress := 40302;
   TCP_Data_Station5[2].Mod_Client[4].modbusDataAddress := 0;
   TCP_Data_Station5[2].Mod_Client[5].modbusDataAddress := 1;
   TCP_Data_Station5[2].Mod_Client[6].modbusDataAddress := 0;
   TCP_Data_Station5[3].Mod_Client[1].modbusDataAddress := 40908;
   TCP_Data_Station5[3].Mod_Client[2].modbusDataAddress := 40001;
   TCP_Data_Station5[3].Mod_Client[3].modbusDataAddress := 40302;
   TCP_Data_Station5[3].Mod_Client[4].modbusDataAddress := 0;
   TCP_Data_Station5[3].Mod_Client[5].modbusDataAddress := 1;
   TCP_Data_Station5[3].Mod_Client[6].modbusDataAddress := 0;
   TCP_Data_Station5[4].Mod_Client[1].modbusDataAddress := 40908;
   TCP_Data_Station5[4].Mod_Client[2].modbusDataAddress := 40001;
   TCP_Data_Station5[4].Mod_Client[3].modbusDataAddress := 40302;
   TCP_Data_Station5[4].Mod_Client[4].modbusDataAddress := 0;
   TCP_Data_Station5[4].Mod_Client[5].modbusDataAddress := 1;
   TCP_Data_Station5[4].Mod_Client[6].modbusDataAddress := 0;
   TCP_Data_Station5[5].Mod_Client[1].modbusDataAddress := 40908;
   TCP_Data_Station5[5].Mod_Client[2].modbusDataAddress := 40001;
   TCP_Data_Station5[5].Mod_Client[3].modbusDataAddress := 40302;
   TCP_Data_Station5[5].Mod_Client[4].modbusDataAddress := 0;
   TCP_Data_Station5[5].Mod_Client[5].modbusDataAddress := 1;
   TCP_Data_Station5[5].Mod_Client[6].modbusDataAddress := 0;
   TCP_Data_Station5[6].Mod_Client[1].modbusDataAddress := 40908;
   TCP_Data_Station5[6].Mod_Client[2].modbusDataAddress := 40001;
   TCP_Data_Station5[6].Mod_Client[3].modbusDataAddress := 40302;
   TCP_Data_Station5[6].Mod_Client[4].modbusDataAddress := 0;
   TCP_Data_Station5[6].Mod_Client[5].modbusDataAddress := 1;
   TCP_Data_Station5[6].Mod_Client[6].modbusDataAddress := 0;
   TCP_Data_Station5[1].Mod_Client[1].modbusDataLen := 1;
   TCP_Data_Station5[1].Mod_Client[2].modbusDataLen := 6;
   TCP_Data_Station5[1].Mod_Client[3].modbusDataLen := 1;
   TCP_Data_Station5[1].Mod_Client[4].modbusDataLen := 0;
   TCP_Data_Station5[1].Mod_Client[5].modbusDataLen := 32;
   TCP_Data_Station5[1].Mod_Client[6].modbusDataLen := 1;
   TCP_Data_Station5[2].Mod_Client[1].modbusDataLen := 1;
   TCP_Data_Station5[2].Mod_Client[2].modbusDataLen := 6;
   TCP_Data_Station5[2].Mod_Client[3].modbusDataLen := 1;
   TCP_Data_Station5[2].Mod_Client[4].modbusDataLen := 0;
   TCP_Data_Station5[2].Mod_Client[5].modbusDataLen := 32;
   TCP_Data_Station5[2].Mod_Client[6].modbusDataLen := 1;
   TCP_Data_Station5[3].Mod_Client[1].modbusDataLen := 1;
   TCP_Data_Station5[3].Mod_Client[2].modbusDataLen := 6;
   TCP_Data_Station5[3].Mod_Client[3].modbusDataLen := 1;
   TCP_Data_Station5[3].Mod_Client[4].modbusDataLen := 0;
   TCP_Data_Station5[3].Mod_Client[5].modbusDataLen := 32;
   TCP_Data_Station5[3].Mod_Client[6].modbusDataLen := 1;
   TCP_Data_Station5[4].Mod_Client[1].modbusDataLen := 1;
   TCP_Data_Station5[4].Mod_Client[2].modbusDataLen := 6;
   TCP_Data_Station5[4].Mod_Client[3].modbusDataLen := 1;
   TCP_Data_Station5[4].Mod_Client[4].modbusDataLen := 0;
   TCP_Data_Station5[4].Mod_Client[5].modbusDataLen := 32;
   TCP_Data_Station5[4].Mod_Client[6].modbusDataLen := 1;
   TCP_Data_Station5[5].Mod_Client[1].modbusDataLen := 1;
   TCP_Data_Station5[5].Mod_Client[2].modbusDataLen := 6;
   TCP_Data_Station5[5].Mod_Client[3].modbusDataLen := 1;
   TCP_Data_Station5[5].Mod_Client[4].modbusDataLen := 0;
   TCP_Data_Station5[5].Mod_Client[5].modbusDataLen := 32;
   TCP_Data_Station5[5].Mod_Client[6].modbusDataLen := 1;
   TCP_Data_Station5[6].Mod_Client[1].modbusDataLen := 1;
   TCP_Data_Station5[6].Mod_Client[2].modbusDataLen := 6;
   TCP_Data_Station5[6].Mod_Client[3].modbusDataLen := 1;
   TCP_Data_Station5[6].Mod_Client[4].modbusDataLen := 0;
   TCP_Data_Station5[6].Mod_Client[5].modbusDataLen := 32;
   TCP_Data_Station5[6].Mod_Client[6].modbusDataLen := 1;
   TCP_Data_CHECK_SCALE_1.Mod_TCP_Connect.connectParamClient.InterfaceId := 64;
   TCP_Data_CHECK_SCALE_1.Mod_TCP_Connect.connectParamClient.ID := 21;
   TCP_Data_CHECK_SCALE_1.Mod_TCP_Connect.connectParamClient.ConnectionType := 16#0B;
   TCP_Data_CHECK_SCALE_1.Mod_TCP_Connect.connectParamClient.ActiveEstablished := true;
   TCP_Data_CHECK_SCALE_1.Mod_TCP_Connect.connectParamClient.RemoteAddress.ADDR[1] := 192;
   TCP_Data_CHECK_SCALE_1.Mod_TCP_Connect.connectParamClient.RemoteAddress.ADDR[2] := 168;
   TCP_Data_CHECK_SCALE_1.Mod_TCP_Connect.connectParamClient.RemoteAddress.ADDR[3] := 0;
   TCP_Data_CHECK_SCALE_1.Mod_TCP_Connect.connectParamClient.RemoteAddress.ADDR[4] := 41;
   TCP_Data_CHECK_SCALE_1.Mod_TCP_Connect.connectParamClient.RemotePort := 502;
   TCP_Data_CHECK_SCALE_1.Mod_TCP_Connect.connectParamClient.LocalPort := 0;
   TCP_Data_CHECK_SCALE_1.Mod_Client[1..6].request := false;
   TCP_Data_CHECK_SCALE_1.Mod_Client[1..6].enable := false;
   TCP_Data_CHECK_SCALE_1.Mod_Client[1..6].disconnect := false;
   TCP_Data_CHECK_SCALE_1.Mod_Client[1..6].done := false;
   TCP_Data_CHECK_SCALE_1.Mod_Client[1..6].busy := false;
   TCP_Data_CHECK_SCALE_1.Mod_Client[1..6].error := false;
   TCP_Data_CHECK_SCALE_1.Mod_Client[1..6].status := 16#0;
   TCP_Data_CHECK_SCALE_1.Mod_Client[1..6].statusSave := 16#0;
   TCP_Data_CHECK_SCALE_1.Mod_Client[1].modbusMode := 1;
   TCP_Data_CHECK_SCALE_1.Mod_Client[2].modbusMode := 0;
   TCP_Data_CHECK_SCALE_1.Mod_Client[3].modbusMode := 1;
   TCP_Data_CHECK_SCALE_1.Mod_Client[4..5].modbusMode := 0;
   TCP_Data_CHECK_SCALE_1.Mod_Client[6].modbusMode := 1;
   TCP_Data_CHECK_SCALE_1.Mod_Client[1].modbusDataAddress := 40908;
   TCP_Data_CHECK_SCALE_1.Mod_Client[2].modbusDataAddress := 40011;
   TCP_Data_CHECK_SCALE_1.Mod_Client[3].modbusDataAddress := 40302;
   TCP_Data_CHECK_SCALE_1.Mod_Client[4].modbusDataAddress := 0;
   TCP_Data_CHECK_SCALE_1.Mod_Client[5].modbusDataAddress := 1;
   TCP_Data_CHECK_SCALE_1.Mod_Client[6].modbusDataAddress := 0;
   TCP_Data_CHECK_SCALE_1.Mod_Client[1].modbusDataLen := 1;
   TCP_Data_CHECK_SCALE_1.Mod_Client[2].modbusDataLen := 10;
   TCP_Data_CHECK_SCALE_1.Mod_Client[3].modbusDataLen := 1;
   TCP_Data_CHECK_SCALE_1.Mod_Client[4].modbusDataLen := 0;
   TCP_Data_CHECK_SCALE_1.Mod_Client[5].modbusDataLen := 32;
   TCP_Data_CHECK_SCALE_1.Mod_Client[6].modbusDataLen := 1;
   TCP_Data_CORRECTION_SCALE.Mod_TCP_Connect.connectParamClient.InterfaceId := 64;
   TCP_Data_CORRECTION_SCALE.Mod_TCP_Connect.connectParamClient.ID := 41;
   TCP_Data_CORRECTION_SCALE.Mod_TCP_Connect.connectParamClient.ConnectionType := 16#0B;
   TCP_Data_CORRECTION_SCALE.Mod_TCP_Connect.connectParamClient.ActiveEstablished := TRUE;
   TCP_Data_CORRECTION_SCALE.Mod_TCP_Connect.connectParamClient.RemoteAddress.ADDR[1] := 192;
   TCP_Data_CORRECTION_SCALE.Mod_TCP_Connect.connectParamClient.RemoteAddress.ADDR[2] := 168;
   TCP_Data_CORRECTION_SCALE.Mod_TCP_Connect.connectParamClient.RemoteAddress.ADDR[3] := 0;
   TCP_Data_CORRECTION_SCALE.Mod_TCP_Connect.connectParamClient.RemoteAddress.ADDR[4] := 41;
   TCP_Data_CORRECTION_SCALE.Mod_TCP_Connect.connectParamClient.RemotePort := 502;
END_DATA_BLOCK

DATA_BLOCK "ALARM_DB"   // DB504
{ S7_Optimized_Access := 'FALSE' }
VERSION : 0.1
// stored: AutoNumber false, DBAccessibleFromOPCUA true, IsOnlyStoredInLoadMemory false, IsWriteProtectedInAS false
   VAR
      COMMON_ALM1 : Word;
      COMMON_ALM2 : Word;
      S1_ALARM1 : Word;
      S1_ALARM2 : Word;
      S2_ALM1 : Word;
      S2_ALM2 : Word;
      S3_ALM1 : Word;
      S3_ALM2 : Word;
      S4_ALARM_STN1 : Word;
      S4_ALARM_STN2 : Word;
      S4_ALARM_STN3 : Word;
      S4_ALARM_STN4 : Word;
      S4_ALARM_STN5 : Word;
      S4_ALARM_STN6 : Word;
      S4_ALARM_STN7 : Word;
      S4_ALARM_STN8 : Word;
      S4_ALARM_STN9 : Word;
      S4_ALARM_STN10 : Word;
      S4_ALARM : Word;
   END_VAR
BEGIN
END_DATA_BLOCK

DATA_BLOCK "ALARM_DB_L2"   // DB505
{ S7_Optimized_Access := 'FALSE' }
VERSION : 0.1
// stored: AutoNumber false, DBAccessibleFromOPCUA true, IsOnlyStoredInLoadMemory false, IsWriteProtectedInAS false
   VAR
      COMMON_ALM1 : Word;
      COMMON_ALM2 : Word;
      S1_ALARM1 : Word;
      S1_ALARM2 : Word;
      S2_ALM1 : Word;
      S2_ALM2 : Word;
      S3_ALM1 : Word;
      S3_ALM2 : Word;
      S5_ALARM_STN1 : Word;
      S5_ALARM_STN2 : Word;
      S5_ALARM_STN3 : Word;
      S5_ALARM_STN4 : Word;
      S5_ALARM_STN5 : Word;
      S5_ALARM_STN6 : Word;
      S5_ALARM_STN7 : Word;
      S5_ALARM_STN8 : Word;
      S5_ALARM_STN9 : Word;
      S5_ALARM_STN10 : Word;
      S5_ALARM : Word;
   END_VAR
BEGIN
END_DATA_BLOCK

DATA_BLOCK "CylinderSetup_DB"   // DB28
{ S7_Optimized_Access := 'FALSE' }
VERSION : 0.1
// stored: AutoNumber true, DBAccessibleFromOPCUA true, IsOnlyStoredInLoadMemory false, IsWriteProtectedInAS false
   VAR
      Array_S1 { S7_SetPoint := 'True'} : Array[1..50] of "uCylinderData";
      Array_S2 { S7_SetPoint := 'True'} : Array[1..50] of "uCylinderData";
      Array_S3 { S7_SetPoint := 'True'} : Array[1..50] of "uCylinderData";
      Array_S4 { S7_SetPoint := 'True'} : Array[1..50] of "uCylinderData";
      Array_S5 { S7_SetPoint := 'True'} : Array[1..50] of "uCylinderData";
      Array_S6 { S7_SetPoint := 'True'} : Array[1..50] of "uCylinderData";
      Array_S7 { S7_SetPoint := 'True'} : Array[1..50] of "uCylinderData";
      Array_S8 { S7_SetPoint := 'True'} : Array[1..50] of "uCylinderData";
      Array_S9 { S7_SetPoint := 'True'} : Array[1..50] of "uCylinderData";
      Array_S10 { S7_SetPoint := 'True'} : Array[1..50] of "uCylinderData";
      Array_S11 { S7_SetPoint := 'True'} : Array[1..50] of "uCylinderData";
      Array_S1_Data : Struct
         Length : Int;
      END_STRUCT;
      Array_S2_Data : Struct
         Length : Int;
      END_STRUCT;
      Array_S3_Data : Struct
         Length : Int;
      END_STRUCT;
      Array_S4_Data : Struct
         Length : Int;
         Array_S2_Data : Struct
            Length : Int;
         END_STRUCT;
      END_STRUCT;
      Array_S5_Data_1 : Struct
         Length : Int;
         Array_S3_Data : Struct
            Length : Int;
         END_STRUCT;
      END_STRUCT;
      "No.OfItems TO S2" : Int := 0;
      Array_R1 { S7_SetPoint := 'True'} : Array[1..50] of "uCylinderData";
      "No.OfItems TO S3" : Int := 0;
      "No.OfItems TO S4" : Int := 0;
      "No.OfItems TO S5" : Int := 0;
      "No.OfItems TO S6" : Int := 1;
      "No.OfItems TO S7" : Int;
      "No.OfItems TO S8" : Int;
      Array_R1_Data : Struct
         Length : Int;
      END_STRUCT;
      Tare_Entry : Real;
   END_VAR
BEGIN
   Array_S6[1].rCylinderID := 0;
   Array_S6[1].rNet_weight := 0.0;
   Array_S6[1].rTareWeight := 0.0;
   Array_S6[1].rGross_Weight := 0.0;
   Array_S6[1].iCylinderType := 0;
END_DATA_BLOCK

DATA_BLOCK "DATA_LOG"   // DB3
{ S7_Optimized_Access := 'TRUE' }
VERSION : 0.1
// stored: AutoNumber true, DBAccessibleFromOPCUA true, IsOnlyStoredInLoadMemory false, IsRetainMemResEnabled false, IsWriteProtectedInAS false, MemoryReserve 100
   VAR
      L1_CY_ID : Int;
      L1_TARE_WT : Real;
      L1_NET_WT : Real;
      L1_GROSS_WT : Real;
      L1_CY_TYPE : Int;
      L2_CY_ID : Int;
      L2_TARE_WT : Real;
      L2_NET_WT : Real;
      L2_GROSS_WT : Real;
      L2_CY_TYPE : Int;
      MALABAR_DOMESTIC_COUNT : Int;
      MALABAR_COMMERCIAL_COUNT : Int;
      BPCL_DOMESTIC_COUNT : Int;
      BPCL_COMMERCIAL_COUNT : Int;
      TOTAL_COUNT : Int;
      L1 { S7_SetPoint := 'True'} : Array[1..6] of "uCylinderData";
      L2 { S7_SetPoint := 'True'} : Array[1..6] of "uCylinderData";
      L1_log_done { S7_SetPoint := 'True'} : Bool;
      L2_log_done : Bool;
      L1_Delet : Bool;
      L2_Delet : Bool;
      "1MINT_BIT" : Bool;
      "1M_BIT" : Bool;
      L1_TOTAL_NET_WT_CY_1 : Real;   // BPCL
      L1_TOTAL_NET_WT_CY_2 : Real;   // MALABAR
      L1_TOTAL_NET_WT_CY_3 : Real;   // BPCL
      L1_TOTAL_NET_WT_CY_4 : Real;   // MALABAR
      L2_TOTAL_NET_WT_CY_1 : Real;
      L2_TOTAL_NET_WT_CY_2 : Real;
      L2_TOTAL_NET_WT_CY_3 : Real;
      L2_TOTAL_NET_WT_CY_4 : Real;
      TOTAL_NET_WT_CY_1_D_BPCL : Real;
      TOTAL_NET_WT_CY_2_C_BPCL : Real;
      TOTAL_NET_WT_CY_3_D_MALA : Real;
      TOTAL_NET_WT_CY_4_C_MALA : Real;
   END_VAR
BEGIN
END_DATA_BLOCK

DATA_BLOCK "Production_report_DB"   // DB2000
{ S7_Optimized_Access := 'FALSE' }
VERSION : 0.1
// stored: AutoNumber false, DBAccessibleFromOPCUA true, IsOnlyStoredInLoadMemory false, IsWriteProtectedInAS false
   VAR
      Production_line_1_Data : Array[1..6] of "uCylinderData";
      Line_1_fill_done { S7_SetPoint := 'True'} : Bool;
      Production_line_2_Data : Array[1..6] of "uCylinderData";
      Line_2_fill_done { S7_SetPoint := 'True'} : Bool;
   END_VAR
BEGIN
END_DATA_BLOCK

DATA_BLOCK "hmi"   // DB27
{ S7_Optimized_Access := 'TRUE' }
VERSION : 0.1
// stored: AutoNumber true, DBAccessibleFromOPCUA true, IsOnlyStoredInLoadMemory false, IsRetainMemResEnabled false, IsWriteProtectedInAS false, MemoryReserve 100
   VAR
      Start : Bool;
      Actual_Weight_cylinder : Real;
      Production_Count : Int;
      Pervious_Day_Count : Int;
      "Cylinder _rejected_S1" : Int;
      Cylinder_Rejected_S6 : Int;
      Truck_No : String;
      Dealer_Code : String;
      Total_Cylinder_Count : Int := 1;
      Domestic_Cylinder_Count : Int;
      Commercial_Cylinder_Count : Int;
      Reset : Bool;
      Cylinder_Count_Actual : Real;
      "Load S1" : Bool;
      "Load S2" : Bool;
      "Load S3" : Bool;
      "Load S4" : Bool;
      "Load S5" : Bool;
      "Load S46" : Bool;
      "Load S56" : Bool;
      "Load S68" : Bool;
      "Load S67" : Bool;
      "Load S78" : Bool;
      Buffer_Reinitialize : Bool;
      cy_t1 : String;
      cy_t2 : String;
      cy_t3 : String;
      cy_t4 : String;
      cy_t5 : String;
      BPCL : Bool;
      MALABAR : Bool;
      In_range : Int;
      "sensing time" : Int;
      password : Int;
      "tare check" : Bool;
      "tare check_1" : Bool;
      "data count" : Int;
      "Load S35" : Bool;
      "Load S56_L2" : Bool;
      "tare check_2" : Bool;
   END_VAR
   VAR RETAIN
      "AUTO/MAN_L1" : Bool;
      "AUTO/MAN_L2" : Bool;
   END_VAR
   VAR
      DIVERTER : Bool;
      NO_itmes_tocopy : Int;
   END_VAR
BEGIN
END_DATA_BLOCK

DATA_BLOCK "hmi_dummy_array"   // DB30
{ S7_Optimized_Access := 'TRUE' }
VERSION : 0.1
// stored: AutoNumber false, DBAccessibleFromOPCUA true, IsOnlyStoredInLoadMemory false, IsRetainMemResEnabled false, IsWriteProtectedInAS false, MemoryReserve 100
   VAR
      array_S1 { S7_SetPoint := 'True'} : Bool;
      array_S2 : Bool;
      S4_PrefillingDummyData { S7_SetPoint := 'True'} : Array[1..10] of "uCylinderData";
      LiftUpFeedback : Array[1..10] of Bool;
      DataransferDone : Bool;
      dummy : "uCylinderData";
      S5_PrefillingdummyData { S7_SetPoint := 'True'} : Array[1..10] of "uCylinderData";
      Gross_Weight { S7_SetPoint := 'True'} : Real;
      hmi_Desicion : Int;
      p_trig : Array[0..5] of Bool;
   END_VAR
BEGIN
   S4_PrefillingDummyData[1..3].iCylinderType := 0;
END_DATA_BLOCK

DATA_BLOCK "real time data"   // DB65
{ S7_Optimized_Access := 'TRUE' }
VERSION : 0.1
// stored: AutoNumber true, DBAccessibleFromOPCUA true, IsOnlyStoredInLoadMemory false, IsRetainMemResEnabled false, IsWriteProtectedInAS false, MemoryReserve 100
   VAR
      "real time data_1" : DTL;
   END_VAR
   VAR RETAIN
      Previous_Day_Count : Int;
   END_VAR
BEGIN
END_DATA_BLOCK

ORGANIZATION_BLOCK "Main"   // OB1, LAD, ProgramCycle
TITLE = "Main Program Sweep (Cycle)"
{ S7_Optimized_Access := 'TRUE' }
VERSION : 0.1
// stored: AutoNumber true, IsIECCheckEnabled false, SetENOAutomatically false
   VAR_INPUT
      Initial_Call : Bool;   // Initial call of this OB
      Remanence : Bool;   // =True, if remanent data are available
   END_VAR
   VAR_TEMP
      temp : Int;
   END_VAR
   VAR_TEMP   // added for the SCL form of the ladder/FBD networks
      _w1 : Bool;
      _w2 : Bool;
      _w3 : Bool;
      _w4 : Bool;
   END_VAR
BEGIN

REGION Network 1
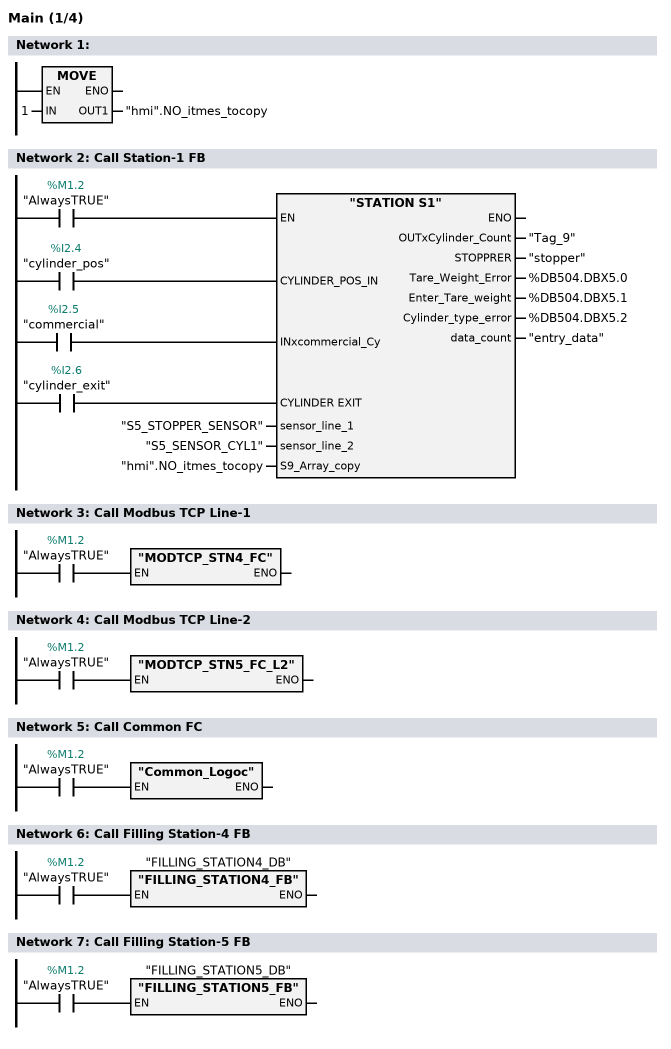
   RUNG wire#powerrail
      Move(in := 1, out1 => "hmi".NO_itmes_tocopy)
   END_RUNG
   // the same network as SCL:
   "hmi".NO_itmes_tocopy := 1;
END_REGION

REGION Network 2: Call Station-1 FB
   RUNG wire#powerrail
      Contact( "AlwaysTRUE" )
      "STATION S1"(CYLINDER_POS_IN := wire#w1, INxcommercial_Cy := wire#w2, "CYLINDER EXIT" := wire#w3, sensor_line_1 := "S5_STOPPER_SENSOR", sensor_line_2 := "S5_SENSOR_CYL1", S9_Array_copy := "hmi".NO_itmes_tocopy, OUTxCylinder_Count => "Tag_9", STOPPRER => "stopper", Tare_Weight_Error => %DB504.DBX5.0, Enter_Tare_weight => %DB504.DBX5.1, Cylinder_type_error => %DB504.DBX5.2, data_count => "entry_data")
   END_RUNG
   RUNG wire#powerrail
      Contact( "cylinder_pos" )
   END_RUNG wire#w1
   RUNG wire#powerrail
      Contact( "commercial" )
   END_RUNG wire#w2
   RUNG wire#powerrail
      Contact( "cylinder_exit" )
   END_RUNG wire#w3
   // the same network as SCL:
   IF "AlwaysTRUE" THEN
       "STATION S1"(CYLINDER_POS_IN := "cylinder_pos",
                    INxcommercial_Cy := "commercial",
                    "CYLINDER EXIT" := "cylinder_exit",
                    sensor_line_1 := "S5_STOPPER_SENSOR",
                    sensor_line_2 := "S5_SENSOR_CYL1",
                    S9_Array_copy := "hmi".NO_itmes_tocopy,
                    OUTxCylinder_Count => "Tag_9",
                    STOPPRER => "stopper",
                    Tare_Weight_Error => %DB504.DBX5.0,
                    Enter_Tare_weight => %DB504.DBX5.1,
                    Cylinder_type_error => %DB504.DBX5.2,
                    data_count => "entry_data");
   END_IF;
END_REGION

REGION Network 3: Call Modbus TCP Line-1
   RUNG wire#powerrail
      Contact( "AlwaysTRUE" )
      "MODTCP_STN4_FC"()
   END_RUNG
   // the same network as SCL:
   IF "AlwaysTRUE" THEN "MODTCP_STN4_FC"(); END_IF;
END_REGION

REGION Network 4: Call Modbus TCP Line-2
   RUNG wire#powerrail
      Contact( "AlwaysTRUE" )
      "MODTCP_STN5_FC_L2"()
   END_RUNG
   // the same network as SCL:
   IF "AlwaysTRUE" THEN "MODTCP_STN5_FC_L2"(); END_IF;
END_REGION

REGION Network 5: Call Common FC
   RUNG wire#powerrail
      Contact( "AlwaysTRUE" )
      "Common_Logoc"()
   END_RUNG
   // the same network as SCL:
   IF "AlwaysTRUE" THEN "Common_Logoc"(); END_IF;
END_REGION

REGION Network 6: Call Filling Station-4 FB
   RUNG wire#powerrail
      Contact( "AlwaysTRUE" )
      "FILLING_STATION4_DB"()
   END_RUNG
   // the same network as SCL:
   IF "AlwaysTRUE" THEN
       "FILLING_STATION4_DB"();   // "FILLING_STATION4_FB"
   END_IF;
END_REGION

REGION Network 7: Call Filling Station-5 FB
   RUNG wire#powerrail
      Contact( "AlwaysTRUE" )
      "FILLING_STATION5_DB"()
   END_RUNG
   // the same network as SCL:
   IF "AlwaysTRUE" THEN
       "FILLING_STATION5_DB"();   // "FILLING_STATION5_FB"
   END_IF;
END_REGION

REGION Network 8
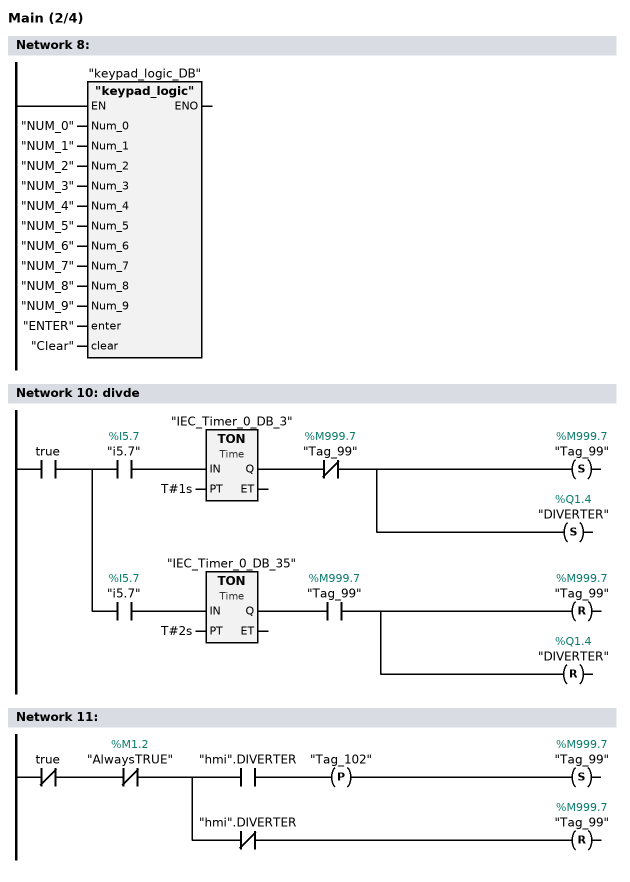
   RUNG wire#powerrail
      "keypad_logic_DB"(Num_0 := "NUM_0", Num_1 := "NUM_1", Num_2 := "NUM_2", Num_3 := "NUM_3", Num_4 := "NUM_4", Num_5 := "NUM_5", Num_6 := "NUM_6", Num_7 := "NUM_7", Num_8 := "NUM_8", Num_9 := "NUM_9", enter := "ENTER", clear := "Clear")
   END_RUNG
   // the same network as SCL:
   "keypad_logic_DB"(Num_0 := "NUM_0",   // "keypad_logic"
                     Num_1 := "NUM_1",
                     Num_2 := "NUM_2",
                     Num_3 := "NUM_3",
                     Num_4 := "NUM_4",
                     Num_5 := "NUM_5",
                     Num_6 := "NUM_6",
                     Num_7 := "NUM_7",
                     Num_8 := "NUM_8",
                     Num_9 := "NUM_9",
                     enter := "ENTER",
                     clear := "Clear");
END_REGION

REGION Network 10: divde
   RUNG wire#powerrail
      Contact( true )
      wire#w1
      Contact( "i5.7" )
      { S7_Templates := "time_type := Time" } "IEC_Timer_0_DB_3".TON(pt := T#1s, et =>)
      I_Contact( "Tag_99" )
      wire#w2
      S_Coil( "Tag_99" )
   END_RUNG
   RUNG wire#w2
      S_Coil( "DIVERTER" )
   END_RUNG
   RUNG wire#w1
      Contact( "i5.7" )
      { S7_Templates := "time_type := Time" } "IEC_Timer_0_DB_35".TON(pt := T#2s, et =>)
      Contact( "Tag_99" )
      wire#w3
      R_Coil( "Tag_99" )
   END_RUNG
   RUNG wire#w3
      R_Coil( "DIVERTER" )
   END_RUNG
   // the same network as SCL:
   "IEC_Timer_0_DB_3".TON(IN := true AND "i5.7", PT := T#1s);
   #_w1 := "IEC_Timer_0_DB_3".Q AND NOT "Tag_99";
   IF #_w1 THEN
       "Tag_99" := TRUE;
       "DIVERTER" := TRUE;
   END_IF;
   "IEC_Timer_0_DB_35".TON(IN := true AND "i5.7", PT := T#2s);
   #_w2 := "IEC_Timer_0_DB_35".Q AND "Tag_99";
   IF #_w2 THEN
       "Tag_99" := FALSE;
       "DIVERTER" := FALSE;
   END_IF;
END_REGION

REGION Network 11
   RUNG wire#powerrail
      I_Contact( true )
      I_Contact( "AlwaysTRUE" )
      wire#w1
      Contact( "hmi".DIVERTER )
      P_Trig( "Tag_102" )
      S_Coil( "Tag_99" )
   END_RUNG
   RUNG wire#w1
      I_Contact( "hmi".DIVERTER )
      R_Coil( "Tag_99" )
   END_RUNG
   // the same network as SCL:
   #_w1 := NOT true AND NOT "AlwaysTRUE";
   #_w2 := #_w1 AND "hmi".DIVERTER;
   #_w3 := #_w2 AND NOT "Tag_102";   // rising edge
   "Tag_102" := #_w2;
   IF #_w3 THEN "Tag_99" := TRUE; END_IF;
   IF #_w1 AND NOT "hmi".DIVERTER THEN "Tag_99" := FALSE; END_IF;
END_REGION

REGION Network 12: DATA LOG L1
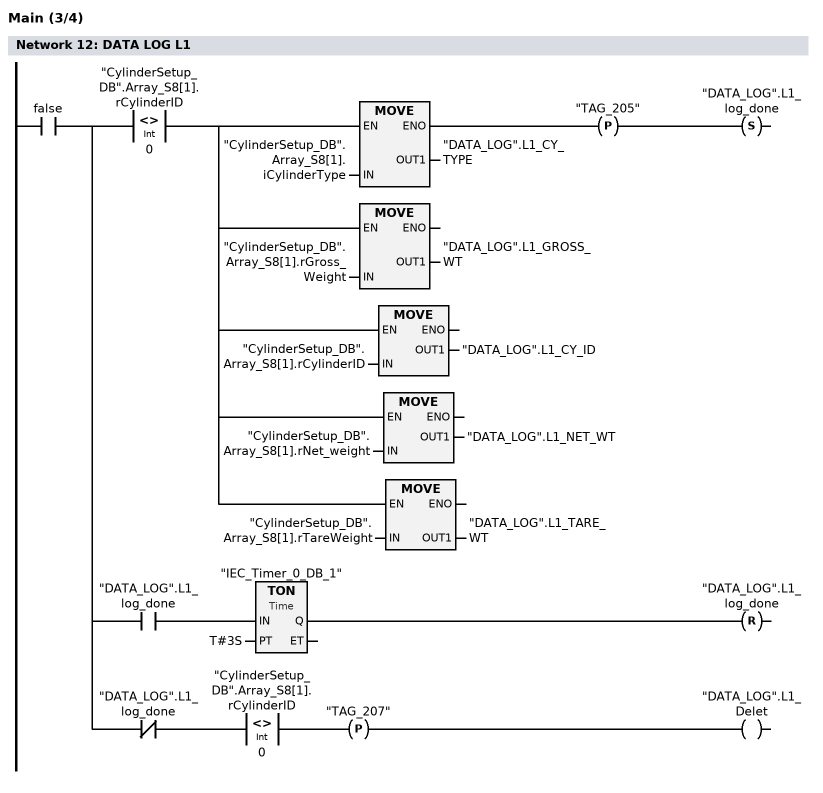
   RUNG wire#powerrail
      Contact( false )
      wire#w1
      { S7_Templates := "SrcType := Int" } NE_Contact(in1 := "CylinderSetup_DB".Array_S8[1].rCylinderID, in2 := 0)
      wire#w2
      Move(in := "CylinderSetup_DB".Array_S8[1].iCylinderType, out1 => "DATA_LOG".L1_CY_TYPE)
      P_Trig( "TAG_205" )
      S_Coil( "DATA_LOG".L1_log_done )
   END_RUNG
   RUNG wire#w2
      Move(in := "CylinderSetup_DB".Array_S8[1].rGross_Weight, out1 => "DATA_LOG".L1_GROSS_WT)
   END_RUNG
   RUNG wire#w2
      Move(in := "CylinderSetup_DB".Array_S8[1].rCylinderID, out1 => "DATA_LOG".L1_CY_ID)
   END_RUNG
   RUNG wire#w2
      Move(in := "CylinderSetup_DB".Array_S8[1].rNet_weight, out1 => "DATA_LOG".L1_NET_WT)
   END_RUNG
   RUNG wire#w2
      Move(in := "CylinderSetup_DB".Array_S8[1].rTareWeight, out1 => "DATA_LOG".L1_TARE_WT)
   END_RUNG
   RUNG wire#w1
      Contact( "DATA_LOG".L1_log_done )
      { S7_Templates := "time_type := Time" } "IEC_Timer_0_DB_1".TON(pt := T#3S, et =>)
      R_Coil( "DATA_LOG".L1_log_done )
   END_RUNG
   RUNG wire#w1
      I_Contact( "DATA_LOG".L1_log_done )
      { S7_Templates := "SrcType := Int" } NE_Contact(in1 := "CylinderSetup_DB".Array_S8[1].rCylinderID, in2 := 0)
      P_Trig( "TAG_207" )
      Coil( "DATA_LOG".L1_Delet )
   END_RUNG
   // the same network as SCL:
   #_w1 := false AND ("CylinderSetup_DB".Array_S8[1].rCylinderID <> 0);
   IF #_w1 THEN "DATA_LOG".L1_CY_TYPE := "CylinderSetup_DB".Array_S8[1].iCylinderType; END_IF;
   #_w2 := #_w1 AND NOT "TAG_205";   // rising edge
   "TAG_205" := #_w1;
   IF #_w2 THEN "DATA_LOG".L1_log_done := TRUE; END_IF;
   IF #_w1 THEN
       "DATA_LOG".L1_GROSS_WT := "CylinderSetup_DB".Array_S8[1].rGross_Weight;
       "DATA_LOG".L1_CY_ID := "CylinderSetup_DB".Array_S8[1].rCylinderID;
       "DATA_LOG".L1_NET_WT := "CylinderSetup_DB".Array_S8[1].rNet_weight;
       "DATA_LOG".L1_TARE_WT := "CylinderSetup_DB".Array_S8[1].rTareWeight;
   END_IF;
   "IEC_Timer_0_DB_1".TON(IN := false AND "DATA_LOG".L1_log_done, PT := T#3S);
   IF "IEC_Timer_0_DB_1".Q THEN "DATA_LOG".L1_log_done := FALSE; END_IF;
   #_w3 := false AND NOT "DATA_LOG".L1_log_done AND ("CylinderSetup_DB".Array_S8[1].rCylinderID <> 0);
   #_w4 := #_w3 AND NOT "TAG_207";   // rising edge
   "TAG_207" := #_w3;
   "DATA_LOG".L1_Delet := #_w4;
END_REGION

REGION Network 13: DATA LOG L2
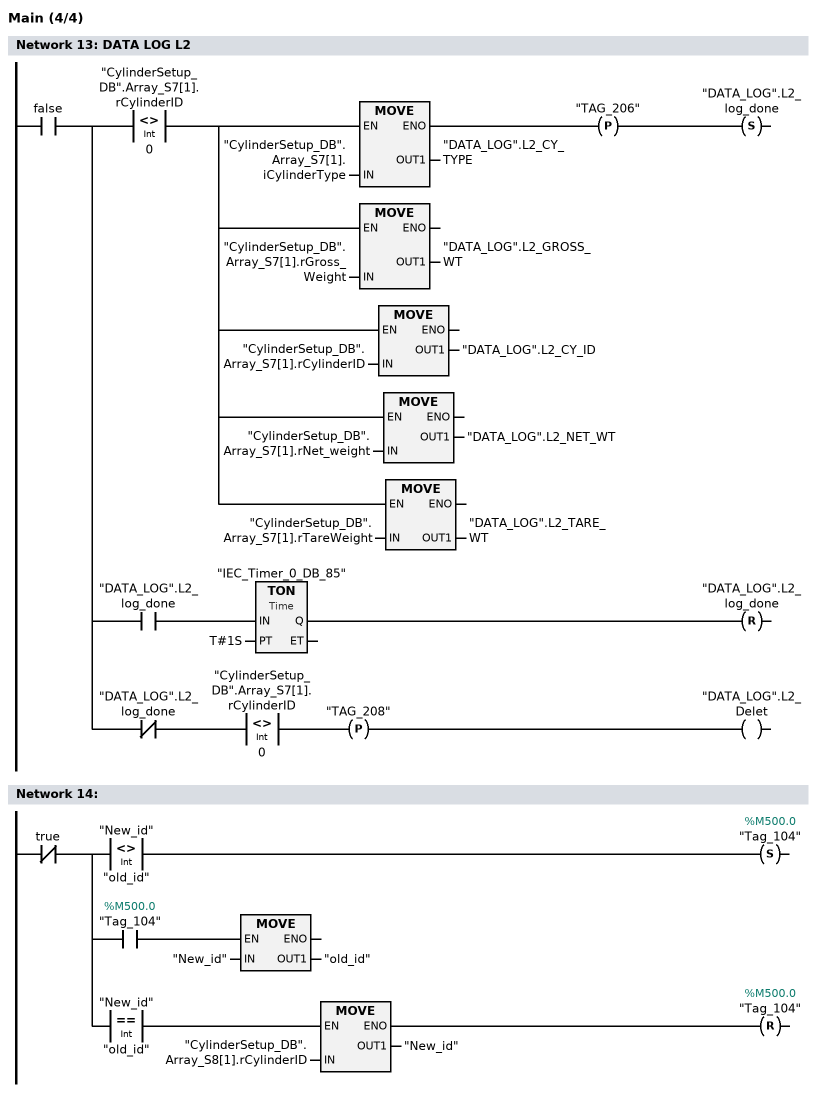
   RUNG wire#powerrail
      Contact( false )
      wire#w1
      { S7_Templates := "SrcType := Int" } NE_Contact(in1 := "CylinderSetup_DB".Array_S7[1].rCylinderID, in2 := 0)
      wire#w2
      Move(in := "CylinderSetup_DB".Array_S7[1].iCylinderType, out1 => "DATA_LOG".L2_CY_TYPE)
      P_Trig( "TAG_206" )
      S_Coil( "DATA_LOG".L2_log_done )
   END_RUNG
   RUNG wire#w2
      Move(in := "CylinderSetup_DB".Array_S7[1].rGross_Weight, out1 => "DATA_LOG".L2_GROSS_WT)
   END_RUNG
   RUNG wire#w2
      Move(in := "CylinderSetup_DB".Array_S7[1].rCylinderID, out1 => "DATA_LOG".L2_CY_ID)
   END_RUNG
   RUNG wire#w2
      Move(in := "CylinderSetup_DB".Array_S7[1].rNet_weight, out1 => "DATA_LOG".L2_NET_WT)
   END_RUNG
   RUNG wire#w2
      Move(in := "CylinderSetup_DB".Array_S7[1].rTareWeight, out1 => "DATA_LOG".L2_TARE_WT)
   END_RUNG
   RUNG wire#w1
      Contact( "DATA_LOG".L2_log_done )
      { S7_Templates := "time_type := Time" } "IEC_Timer_0_DB_85".TON(pt := T#1S, et =>)
      R_Coil( "DATA_LOG".L2_log_done )
   END_RUNG
   RUNG wire#w1
      I_Contact( "DATA_LOG".L2_log_done )
      { S7_Templates := "SrcType := Int" } NE_Contact(in1 := "CylinderSetup_DB".Array_S7[1].rCylinderID, in2 := 0)
      P_Trig( "TAG_208" )
      Coil( "DATA_LOG".L2_Delet )
   END_RUNG
   // the same network as SCL:
   #_w1 := false AND ("CylinderSetup_DB".Array_S7[1].rCylinderID <> 0);
   IF #_w1 THEN "DATA_LOG".L2_CY_TYPE := "CylinderSetup_DB".Array_S7[1].iCylinderType; END_IF;
   #_w2 := #_w1 AND NOT "TAG_206";   // rising edge
   "TAG_206" := #_w1;
   IF #_w2 THEN "DATA_LOG".L2_log_done := TRUE; END_IF;
   IF #_w1 THEN
       "DATA_LOG".L2_GROSS_WT := "CylinderSetup_DB".Array_S7[1].rGross_Weight;
       "DATA_LOG".L2_CY_ID := "CylinderSetup_DB".Array_S7[1].rCylinderID;
       "DATA_LOG".L2_NET_WT := "CylinderSetup_DB".Array_S7[1].rNet_weight;
       "DATA_LOG".L2_TARE_WT := "CylinderSetup_DB".Array_S7[1].rTareWeight;
   END_IF;
   "IEC_Timer_0_DB_85".TON(IN := false AND "DATA_LOG".L2_log_done, PT := T#1S);
   IF "IEC_Timer_0_DB_85".Q THEN "DATA_LOG".L2_log_done := FALSE; END_IF;
   #_w3 := false AND NOT "DATA_LOG".L2_log_done AND ("CylinderSetup_DB".Array_S7[1].rCylinderID <> 0);
   #_w4 := #_w3 AND NOT "TAG_208";   // rising edge
   "TAG_208" := #_w3;
   "DATA_LOG".L2_Delet := #_w4;
END_REGION

REGION Network 14
   RUNG wire#powerrail
      I_Contact( true )
      wire#w1
      { S7_Templates := "SrcType := Int" } NE_Contact(in1 := "New_id", in2 := "old_id")
      S_Coil( "Tag_104" )
   END_RUNG
   RUNG wire#w1
      Contact( "Tag_104" )
      Move(in := "New_id", out1 => "old_id")
   END_RUNG
   RUNG wire#w1
      { S7_Templates := "SrcType := Int" } EQ_Contact(in1 := "New_id", in2 := "old_id")
      Move(in := "CylinderSetup_DB".Array_S8[1].rCylinderID, out1 => "New_id")
      R_Coil( "Tag_104" )
   END_RUNG
   // the same network as SCL:
   IF NOT true AND ("New_id" <> "old_id") THEN "Tag_104" := TRUE; END_IF;
   IF NOT true AND "Tag_104" THEN "old_id" := "New_id"; END_IF;
   #_w1 := NOT true AND ("New_id" = "old_id");
   IF #_w1 THEN
       "New_id" := "CylinderSetup_DB".Array_S8[1].rCylinderID;
       "Tag_104" := FALSE;
   END_IF;
END_REGION
END_ORGANIZATION_BLOCK

FUNCTION "STATION S1" : Void   // FC3, LAD
{ S7_Optimized_Access := 'TRUE' }
VERSION : 0.1
// stored: AutoNumber true, IsIECCheckEnabled false, SetENOAutomatically false, UDAEnableTagReadback false
   VAR_INPUT
      CYLINDER_POS_IN : Bool;
      INxcommercial_Cy : Bool;
      "CYLINDER EXIT" : Bool;
      sensor_line_1 : Bool;
      sensor_line_2 : Bool;
   END_VAR
   VAR_OUTPUT
      OUTxCylinder_Count : Bool;
      STOPPRER : Bool;
      Tare_Weight_Error : Bool;
      Enter_Tare_weight : Bool;
      Cylinder_type_error : Bool;
      data_count : Int;
   END_VAR
   VAR_IN_OUT
      S9_Array_copy : Int;
   END_VAR
   VAR_TEMP
      TRUCK : String;
      Start : Bool;
      copied_item : Int;
      Ret_val_1 : Int;
      Out_RD : DTL;
      Difference_Domestic_Cy : Real;
      Difference_commercial_Cy : Real;
      set_bit : Bool;
      Full_Wieght_Difference : Real;
      idx1 : Int;
      idx2 : Int;
      idx3 : Int;
      idx4 : Int;
      idx5 : Int;
      idx6 : Int;
      idx7 : Int;
      Gross_Weight : Real;
      "cylinder ok" : Bool;
      ptrig : Bool;
      ptrig_1 : Bool;
      ptrig_2 : Bool;
      TEMP : Int;
      pass : Bool;
      FILL_DB : Bool;
      TEMP_1 : Int;
      TEMP_2 : Int;
      TEMP_3 : Int;
      TEMP_4 : Int;
      TEMP_5 : Int;
      TEMP_6 : Int;
      TEMP_7 : Int;
      TEMP_8 : Int;
      TEMP_9 : Int;
      TEMP_10 : Int;
      TEMP_11 : Int;
      TEMP_12 : Int;
      TEMP_13 : Int;
      TEMP_14 : Int;
   END_VAR
   VAR_TEMP   // added for the SCL form of the ladder/FBD networks
      _w1 : Bool;
      _w2 : Bool;
      _w3 : Bool;
      _w4 : Bool;
      _w5 : Bool;
      _w6 : Bool;
      _w7 : Bool;
      _w8 : Bool;
      _w9 : Bool;
   END_VAR
BEGIN

REGION Network 1: Cylinder_Count
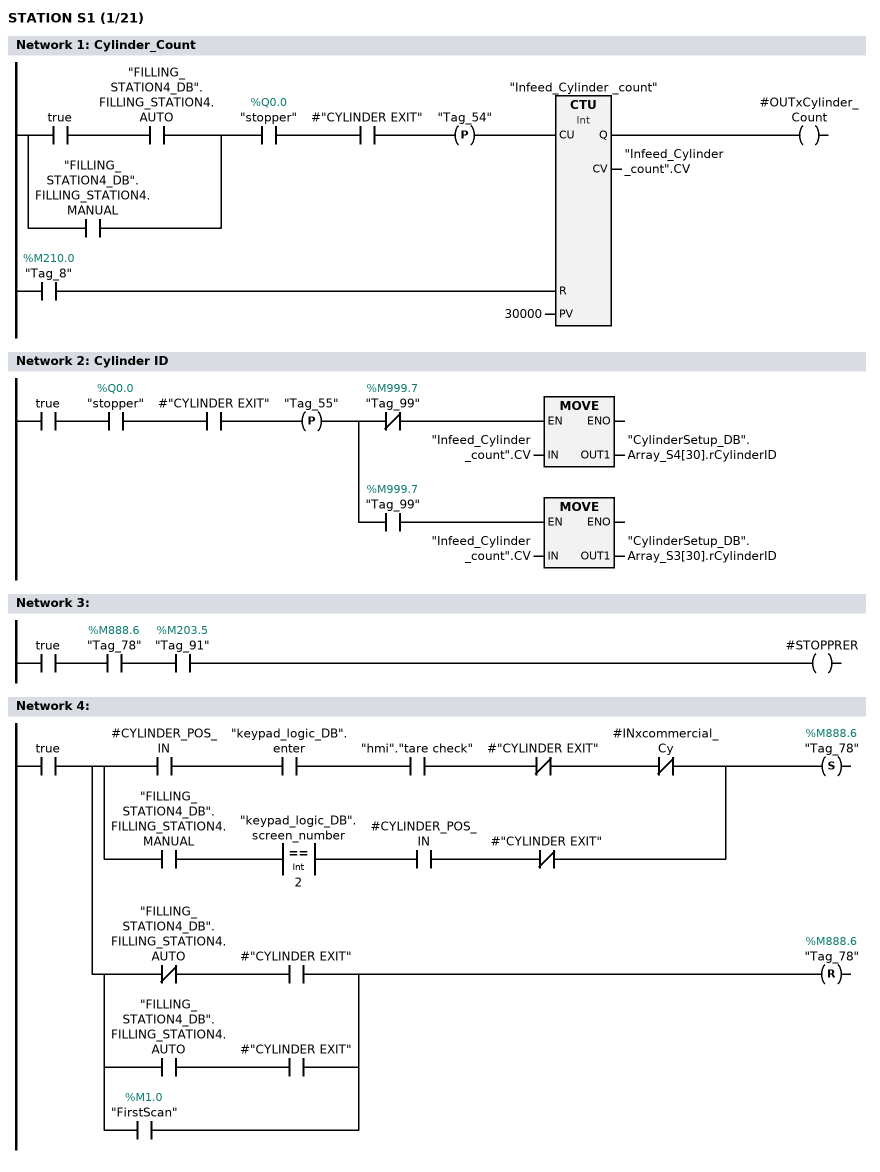
   RUNG wire#powerrail
      Contact( true )
      Contact( "FILLING_STATION4_DB".FILLING_STATION4.AUTO )
      wire#w1
      Contact( "stopper" )
      Contact( #"CYLINDER EXIT" )
      P_Trig( "Tag_54" )
      { S7_Templates := "value_type := Int" } "Infeed_Cylinder _count".CTU(r := wire#w2, pv := 30000, cv => "Infeed_Cylinder _count".CV)
      Coil( #OUTxCylinder_Count )
   END_RUNG
   RUNG wire#powerrail
      Contact( "FILLING_STATION4_DB".FILLING_STATION4.MANUAL )
   END_RUNG wire#w1
   RUNG wire#powerrail
      Contact( "Tag_8" )
   END_RUNG wire#w2
   // the same network as SCL:
   #_w1 := ((true AND "FILLING_STATION4_DB".FILLING_STATION4.AUTO) OR "FILLING_STATION4_DB".FILLING_STATION4.MANUAL) AND "stopper" AND #"CYLINDER EXIT";
   #_w2 := #_w1 AND NOT "Tag_54";   // rising edge
   "Tag_54" := #_w1;
   "Infeed_Cylinder _count".CTU(CU := #_w2, R := "Tag_8", PV := 30000, CV => "Infeed_Cylinder _count".CV);
   #OUTxCylinder_Count := "Infeed_Cylinder _count".Q;
END_REGION

REGION Network 2: Cylinder ID
   RUNG wire#powerrail
      Contact( true )
      Contact( "stopper" )
      Contact( #"CYLINDER EXIT" )
      P_Trig( "Tag_55" )
      wire#w1
      I_Contact( "Tag_99" )
      Move(in := "Infeed_Cylinder _count".CV, out1 => "CylinderSetup_DB".Array_S4[30].rCylinderID)
   END_RUNG
   RUNG wire#w1
      Contact( "Tag_99" )
      Move(in := "Infeed_Cylinder _count".CV, out1 => "CylinderSetup_DB".Array_S3[30].rCylinderID)
   END_RUNG
   // the same network as SCL:
   #_w1 := true AND "stopper" AND #"CYLINDER EXIT";
   #_w2 := #_w1 AND NOT "Tag_55";   // rising edge
   "Tag_55" := #_w1;
   IF #_w2 AND NOT "Tag_99" THEN
       "CylinderSetup_DB".Array_S4[30].rCylinderID := "Infeed_Cylinder _count".CV;
   END_IF;
   IF #_w2 AND "Tag_99" THEN
       "CylinderSetup_DB".Array_S3[30].rCylinderID := "Infeed_Cylinder _count".CV;
   END_IF;
END_REGION

REGION Network 3
   RUNG wire#powerrail
      Contact( true )
      Contact( "Tag_78" )
      Contact( "Tag_91" )
      Coil( #STOPPRER )
   END_RUNG
   // the same network as SCL:
   #STOPPRER := true AND "Tag_78" AND "Tag_91";
END_REGION

REGION Network 4
   RUNG wire#powerrail
      Contact( true )
      wire#w1
      Contact( #CYLINDER_POS_IN )
      Contact( "keypad_logic_DB".enter )
      Contact( "hmi"."tare check" )
      I_Contact( #"CYLINDER EXIT" )
      I_Contact( #INxcommercial_Cy )
      wire#w2
      S_Coil( "Tag_78" )
   END_RUNG
   RUNG wire#w1
      Contact( "FILLING_STATION4_DB".FILLING_STATION4.MANUAL )
      { S7_Templates := "SrcType := Int" } EQ_Contact(in1 := "keypad_logic_DB".screen_number, in2 := 2)
      Contact( #CYLINDER_POS_IN )
      I_Contact( #"CYLINDER EXIT" )
   END_RUNG wire#w2
   RUNG wire#w1
      I_Contact( "FILLING_STATION4_DB".FILLING_STATION4.AUTO )
      Contact( #"CYLINDER EXIT" )
      wire#w3
      R_Coil( "Tag_78" )
   END_RUNG
   RUNG wire#w1
      Contact( "FILLING_STATION4_DB".FILLING_STATION4.AUTO )
      Contact( #"CYLINDER EXIT" )
   END_RUNG wire#w3
   RUNG wire#w1
      Contact( "FirstScan" )
   END_RUNG wire#w3
   // the same network as SCL:
   IF true AND ((#CYLINDER_POS_IN AND "keypad_logic_DB".enter AND "hmi"."tare check" AND NOT #"CYLINDER EXIT" AND NOT #INxcommercial_Cy) OR ("FILLING_STATION4_DB".FILLING_STATION4.MANUAL AND ("keypad_logic_DB".screen_number = 2) AND #CYLINDER_POS_IN AND NOT #"CYLINDER EXIT")) THEN
       "Tag_78" := TRUE;
   END_IF;
   IF true AND ((NOT "FILLING_STATION4_DB".FILLING_STATION4.AUTO AND #"CYLINDER EXIT") OR ("FILLING_STATION4_DB".FILLING_STATION4.AUTO AND #"CYLINDER EXIT") OR "FirstScan") THEN
       "Tag_78" := FALSE;
   END_IF;
END_REGION

REGION Network 5: Domestic_Cylinder_Details
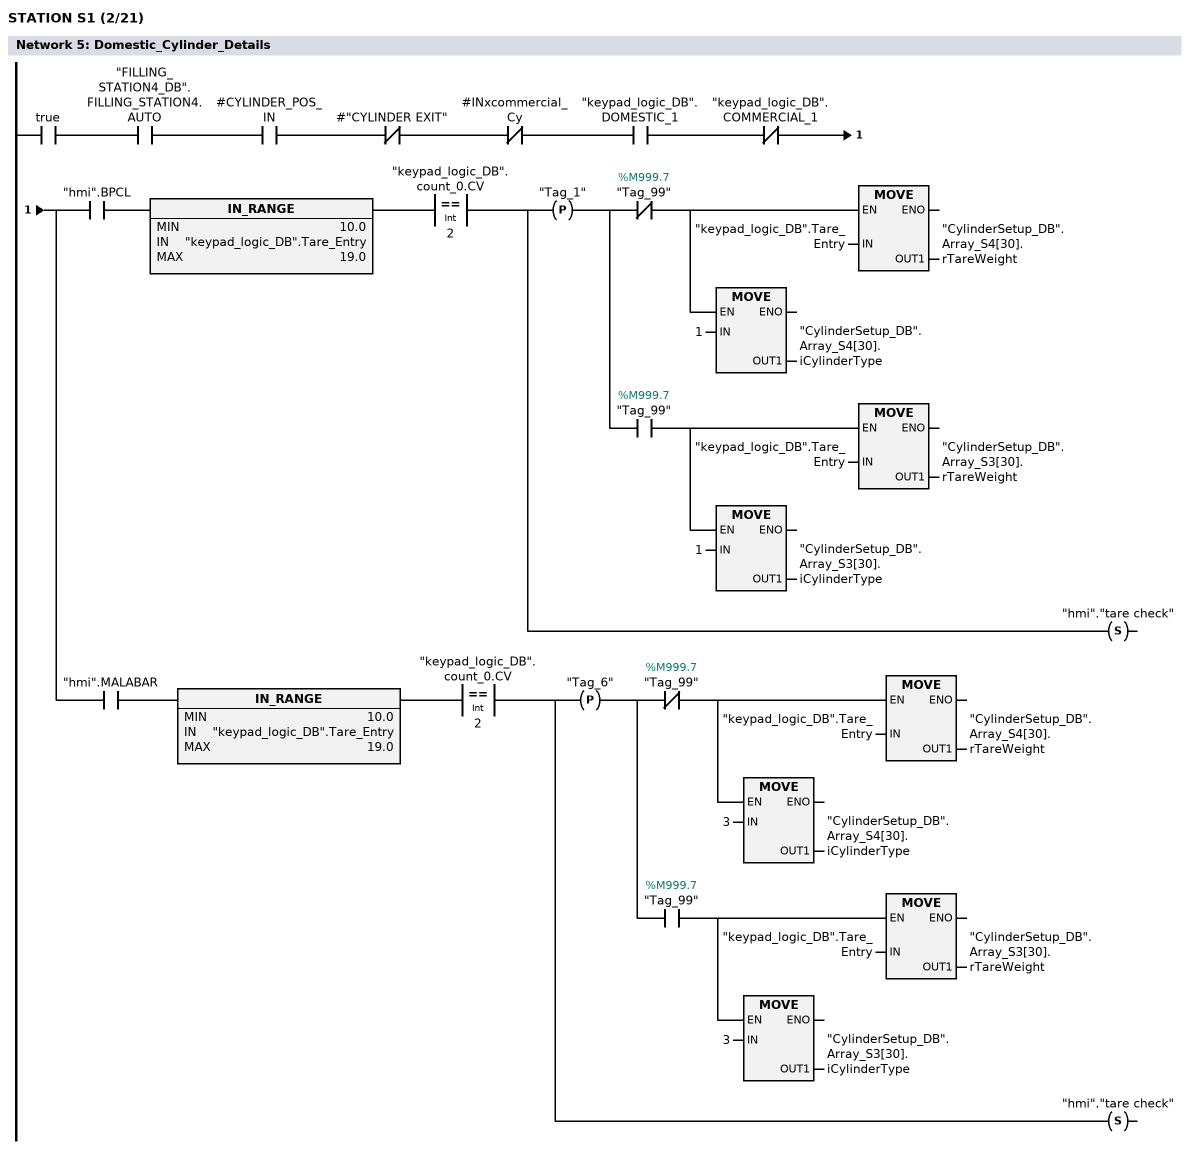
   RUNG wire#powerrail
      Contact( true )
      Contact( "FILLING_STATION4_DB".FILLING_STATION4.AUTO )
      Contact( #CYLINDER_POS_IN )
      I_Contact( #"CYLINDER EXIT" )
      I_Contact( #INxcommercial_Cy )
      Contact( "keypad_logic_DB".DOMESTIC_1 )
      I_Contact( "keypad_logic_DB".COMMERCIAL_1 )
      wire#w1
      Contact( "hmi".BPCL )
      { S7_Templates := "SrcType := Real" } InRange(min := 10.0, in := "keypad_logic_DB".Tare_Entry, max := 19.0)
      { S7_Templates := "SrcType := Int" } EQ_Contact(in1 := "keypad_logic_DB".count_0.CV, in2 := 2)
      wire#w2
      P_Trig( "Tag_1" )
      wire#w3
      I_Contact( "Tag_99" )
      wire#w4
      Move(in := "keypad_logic_DB".Tare_Entry, out1 => "CylinderSetup_DB".Array_S4[30].rTareWeight)
   END_RUNG
   RUNG wire#w4
      Move(in := 1, out1 => "CylinderSetup_DB".Array_S4[30].iCylinderType)
   END_RUNG
   RUNG wire#w3
      Contact( "Tag_99" )
      wire#w5
      Move(in := "keypad_logic_DB".Tare_Entry, out1 => "CylinderSetup_DB".Array_S3[30].rTareWeight)
   END_RUNG
   RUNG wire#w5
      Move(in := 1, out1 => "CylinderSetup_DB".Array_S3[30].iCylinderType)
   END_RUNG
   RUNG wire#w2
      S_Coil( "hmi"."tare check" )
   END_RUNG
   RUNG wire#w1
      Contact( "hmi".MALABAR )
      { S7_Templates := "SrcType := Real" } InRange(min := 10.0, in := "keypad_logic_DB".Tare_Entry, max := 19.0)
      { S7_Templates := "SrcType := Int" } EQ_Contact(in1 := "keypad_logic_DB".count_0.CV, in2 := 2)
      wire#w6
      P_Trig( "Tag_6" )
      wire#w7
      I_Contact( "Tag_99" )
      wire#w8
      Move(in := "keypad_logic_DB".Tare_Entry, out1 => "CylinderSetup_DB".Array_S4[30].rTareWeight)
   END_RUNG
   RUNG wire#w8
      Move(in := 3, out1 => "CylinderSetup_DB".Array_S4[30].iCylinderType)
   END_RUNG
   RUNG wire#w7
      Contact( "Tag_99" )
      wire#w9
      Move(in := "keypad_logic_DB".Tare_Entry, out1 => "CylinderSetup_DB".Array_S3[30].rTareWeight)
   END_RUNG
   RUNG wire#w9
      Move(in := 3, out1 => "CylinderSetup_DB".Array_S3[30].iCylinderType)
   END_RUNG
   RUNG wire#w6
      S_Coil( "hmi"."tare check" )
   END_RUNG
   // the same network as SCL:
   #_w1 := true AND "FILLING_STATION4_DB".FILLING_STATION4.AUTO AND #CYLINDER_POS_IN AND NOT #"CYLINDER EXIT" AND NOT #INxcommercial_Cy AND "keypad_logic_DB".DOMESTIC_1 AND NOT "keypad_logic_DB".COMMERCIAL_1;
   #_w2 := #_w1 AND "hmi".BPCL AND (10.0 <= "keypad_logic_DB".Tare_Entry) AND ("keypad_logic_DB".Tare_Entry <= 19.0) AND ("keypad_logic_DB".count_0.CV = 2);
   #_w3 := #_w2 AND NOT "Tag_1";   // rising edge
   "Tag_1" := #_w2;
   IF #_w3 AND NOT "Tag_99" THEN
       "CylinderSetup_DB".Array_S4[30].rTareWeight := "keypad_logic_DB".Tare_Entry;
       "CylinderSetup_DB".Array_S4[30].iCylinderType := 1;
   END_IF;
   IF #_w3 AND "Tag_99" THEN
       "CylinderSetup_DB".Array_S3[30].rTareWeight := "keypad_logic_DB".Tare_Entry;
       "CylinderSetup_DB".Array_S3[30].iCylinderType := 1;
   END_IF;
   IF #_w2 THEN "hmi"."tare check" := TRUE; END_IF;
   #_w4 := #_w1 AND "hmi".MALABAR AND (10.0 <= "keypad_logic_DB".Tare_Entry) AND ("keypad_logic_DB".Tare_Entry <= 19.0) AND ("keypad_logic_DB".count_0.CV = 2);
   #_w5 := #_w4 AND NOT "Tag_6";   // rising edge
   "Tag_6" := #_w4;
   IF #_w5 AND NOT "Tag_99" THEN
       "CylinderSetup_DB".Array_S4[30].rTareWeight := "keypad_logic_DB".Tare_Entry;
       "CylinderSetup_DB".Array_S4[30].iCylinderType := 3;
   END_IF;
   IF #_w5 AND "Tag_99" THEN
       "CylinderSetup_DB".Array_S3[30].rTareWeight := "keypad_logic_DB".Tare_Entry;
       "CylinderSetup_DB".Array_S3[30].iCylinderType := 3;
   END_IF;
   IF #_w4 THEN "hmi"."tare check" := TRUE; END_IF;
END_REGION

REGION Network 6: DOMESTIC_ALARM
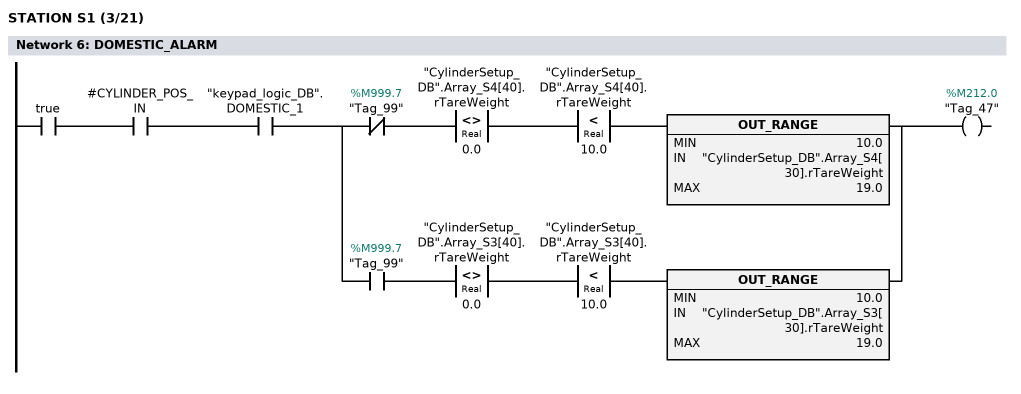
   "Tag_47" := true AND #CYLINDER_POS_IN AND "keypad_logic_DB".DOMESTIC_1 AND ((NOT "Tag_99" AND ("CylinderSetup_DB".Array_S4[40].rTareWeight <> 0.0) AND ("CylinderSetup_DB".Array_S4[40].rTareWeight < 10.0) AND (("CylinderSetup_DB".Array_S4[30].rTareWeight < 10.0) OR ("CylinderSetup_DB".Array_S4[30].rTareWeight > 19.0))) OR ("Tag_99" AND ("CylinderSetup_DB".Array_S3[40].rTareWeight <> 0.0) AND ("CylinderSetup_DB".Array_S3[40].rTareWeight < 10.0) AND (("CylinderSetup_DB".Array_S3[30].rTareWeight < 10.0) OR ("CylinderSetup_DB".Array_S3[30].rTareWeight > 19.0))));
END_REGION

REGION Network 7: Commercial_Cylinder_Details
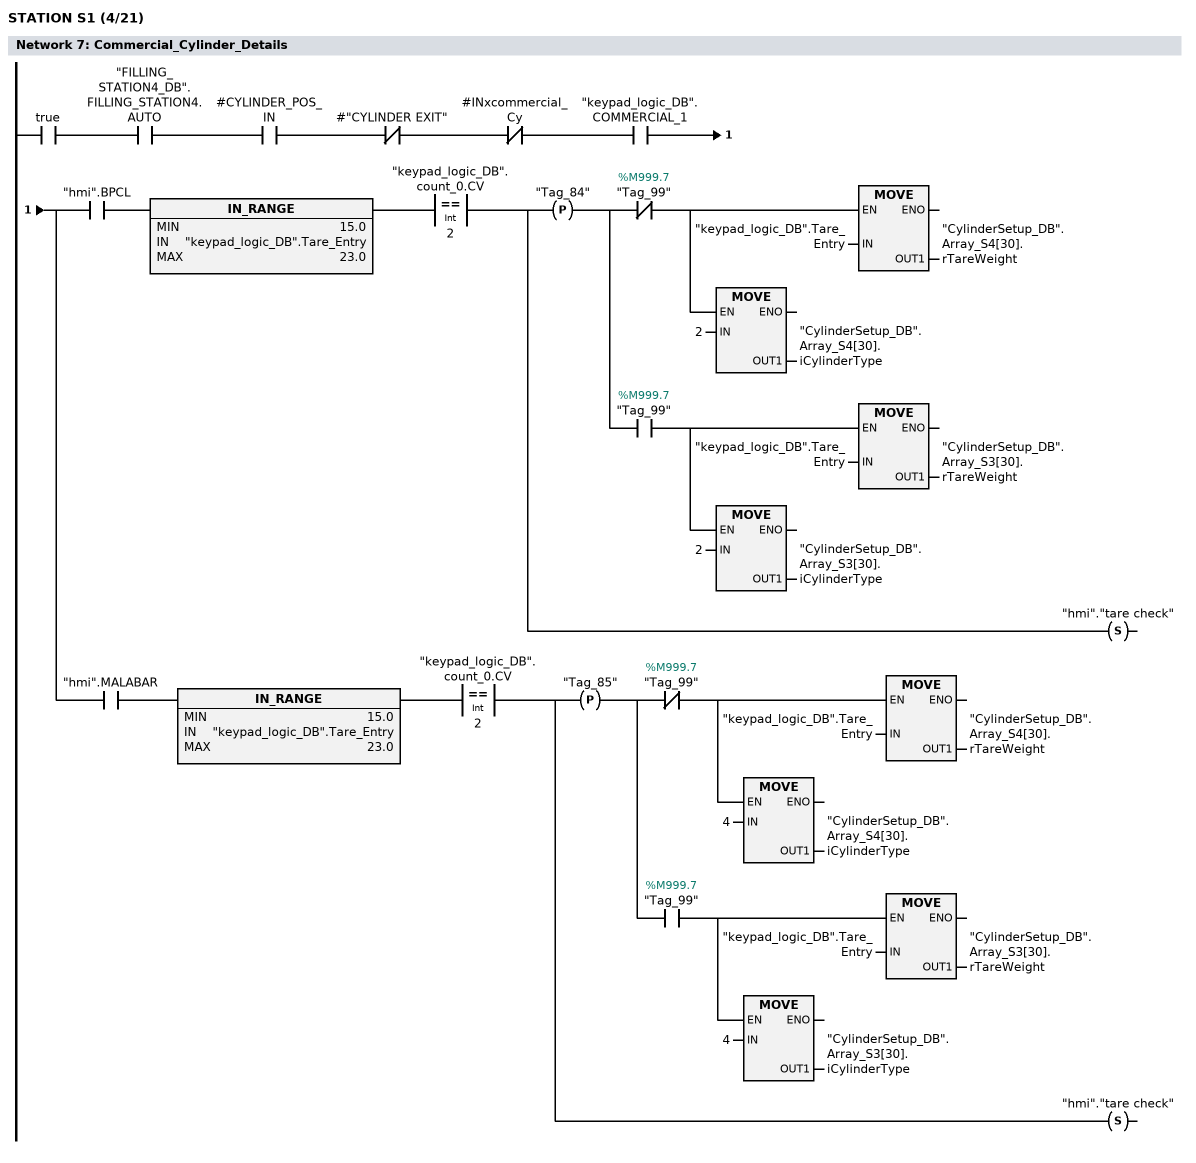
   RUNG wire#powerrail
      Contact( true )
      Contact( "FILLING_STATION4_DB".FILLING_STATION4.AUTO )
      Contact( #CYLINDER_POS_IN )
      I_Contact( #"CYLINDER EXIT" )
      I_Contact( #INxcommercial_Cy )
      Contact( "keypad_logic_DB".COMMERCIAL_1 )
      wire#w1
      Contact( "hmi".BPCL )
      { S7_Templates := "SrcType := Real" } InRange(min := 15.0, in := "keypad_logic_DB".Tare_Entry, max := 23.0)
      { S7_Templates := "SrcType := Int" } EQ_Contact(in1 := "keypad_logic_DB".count_0.CV, in2 := 2)
      wire#w2
      P_Trig( "Tag_84" )
      wire#w3
      I_Contact( "Tag_99" )
      wire#w4
      Move(in := "keypad_logic_DB".Tare_Entry, out1 => "CylinderSetup_DB".Array_S4[30].rTareWeight)
   END_RUNG
   RUNG wire#w4
      Move(in := 2, out1 => "CylinderSetup_DB".Array_S4[30].iCylinderType)
   END_RUNG
   RUNG wire#w3
      Contact( "Tag_99" )
      wire#w5
      Move(in := "keypad_logic_DB".Tare_Entry, out1 => "CylinderSetup_DB".Array_S3[30].rTareWeight)
   END_RUNG
   RUNG wire#w5
      Move(in := 2, out1 => "CylinderSetup_DB".Array_S3[30].iCylinderType)
   END_RUNG
   RUNG wire#w2
      S_Coil( "hmi"."tare check" )
   END_RUNG
   RUNG wire#w1
      Contact( "hmi".MALABAR )
      { S7_Templates := "SrcType := Real" } InRange(min := 15.0, in := "keypad_logic_DB".Tare_Entry, max := 23.0)
      { S7_Templates := "SrcType := Int" } EQ_Contact(in1 := "keypad_logic_DB".count_0.CV, in2 := 2)
      wire#w6
      P_Trig( "Tag_85" )
      wire#w7
      I_Contact( "Tag_99" )
      wire#w8
      Move(in := "keypad_logic_DB".Tare_Entry, out1 => "CylinderSetup_DB".Array_S4[30].rTareWeight)
   END_RUNG
   RUNG wire#w8
      Move(in := 4, out1 => "CylinderSetup_DB".Array_S4[30].iCylinderType)
   END_RUNG
   RUNG wire#w7
      Contact( "Tag_99" )
      wire#w9
      Move(in := "keypad_logic_DB".Tare_Entry, out1 => "CylinderSetup_DB".Array_S3[30].rTareWeight)
   END_RUNG
   RUNG wire#w9
      Move(in := 4, out1 => "CylinderSetup_DB".Array_S3[30].iCylinderType)
   END_RUNG
   RUNG wire#w6
      S_Coil( "hmi"."tare check" )
   END_RUNG
   // the same network as SCL:
   #_w1 := true AND "FILLING_STATION4_DB".FILLING_STATION4.AUTO AND #CYLINDER_POS_IN AND NOT #"CYLINDER EXIT" AND NOT #INxcommercial_Cy AND "keypad_logic_DB".COMMERCIAL_1;
   #_w2 := #_w1 AND "hmi".BPCL AND (15.0 <= "keypad_logic_DB".Tare_Entry) AND ("keypad_logic_DB".Tare_Entry <= 23.0) AND ("keypad_logic_DB".count_0.CV = 2);
   #_w3 := #_w2 AND NOT "Tag_84";   // rising edge
   "Tag_84" := #_w2;
   IF #_w3 AND NOT "Tag_99" THEN
       "CylinderSetup_DB".Array_S4[30].rTareWeight := "keypad_logic_DB".Tare_Entry;
       "CylinderSetup_DB".Array_S4[30].iCylinderType := 2;
   END_IF;
   IF #_w3 AND "Tag_99" THEN
       "CylinderSetup_DB".Array_S3[30].rTareWeight := "keypad_logic_DB".Tare_Entry;
       "CylinderSetup_DB".Array_S3[30].iCylinderType := 2;
   END_IF;
   IF #_w2 THEN "hmi"."tare check" := TRUE; END_IF;
   #_w4 := #_w1 AND "hmi".MALABAR AND (15.0 <= "keypad_logic_DB".Tare_Entry) AND ("keypad_logic_DB".Tare_Entry <= 23.0) AND ("keypad_logic_DB".count_0.CV = 2);
   #_w5 := #_w4 AND NOT "Tag_85";   // rising edge
   "Tag_85" := #_w4;
   IF #_w5 AND NOT "Tag_99" THEN
       "CylinderSetup_DB".Array_S4[30].rTareWeight := "keypad_logic_DB".Tare_Entry;
       "CylinderSetup_DB".Array_S4[30].iCylinderType := 4;
   END_IF;
   IF #_w5 AND "Tag_99" THEN
       "CylinderSetup_DB".Array_S3[30].rTareWeight := "keypad_logic_DB".Tare_Entry;
       "CylinderSetup_DB".Array_S3[30].iCylinderType := 4;
   END_IF;
   IF #_w4 THEN "hmi"."tare check" := TRUE; END_IF;
END_REGION

REGION Network 8: COMMERCIAL_ALARM
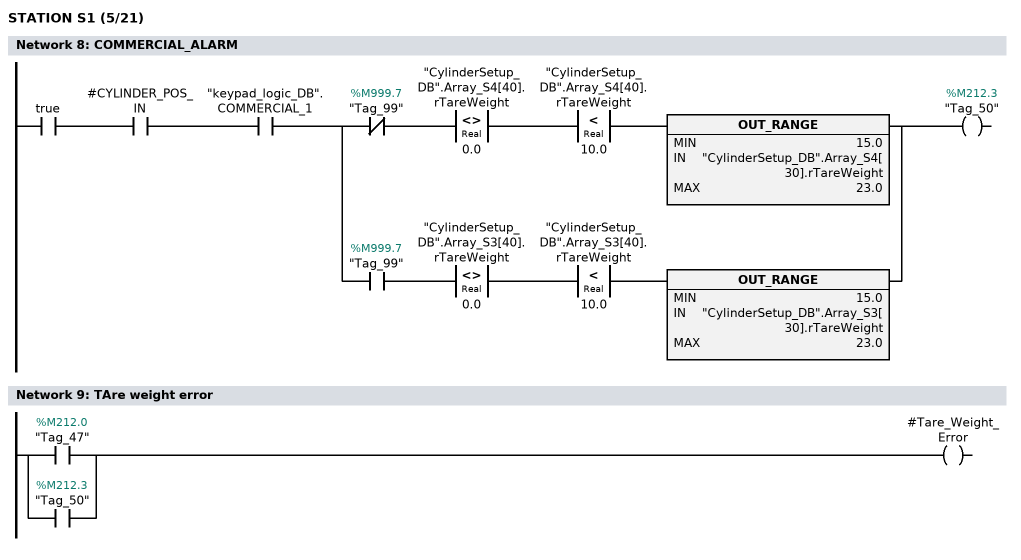
   "Tag_50" := true AND #CYLINDER_POS_IN AND "keypad_logic_DB".COMMERCIAL_1 AND ((NOT "Tag_99" AND ("CylinderSetup_DB".Array_S4[40].rTareWeight <> 0.0) AND ("CylinderSetup_DB".Array_S4[40].rTareWeight < 10.0) AND (("CylinderSetup_DB".Array_S4[30].rTareWeight < 15.0) OR ("CylinderSetup_DB".Array_S4[30].rTareWeight > 23.0))) OR ("Tag_99" AND ("CylinderSetup_DB".Array_S3[40].rTareWeight <> 0.0) AND ("CylinderSetup_DB".Array_S3[40].rTareWeight < 10.0) AND (("CylinderSetup_DB".Array_S3[30].rTareWeight < 15.0) OR ("CylinderSetup_DB".Array_S3[30].rTareWeight > 23.0))));
END_REGION

REGION Network 9: TAre weight error
   RUNG wire#powerrail
      Contact( "Tag_47" )
      wire#w1
      Coil( #Tare_Weight_Error )
   END_RUNG
   RUNG wire#powerrail
      Contact( "Tag_50" )
   END_RUNG wire#w1
   // the same network as SCL:
   #Tare_Weight_Error := "Tag_47" OR "Tag_50";
END_REGION

REGION Network 10: S4_Array Move
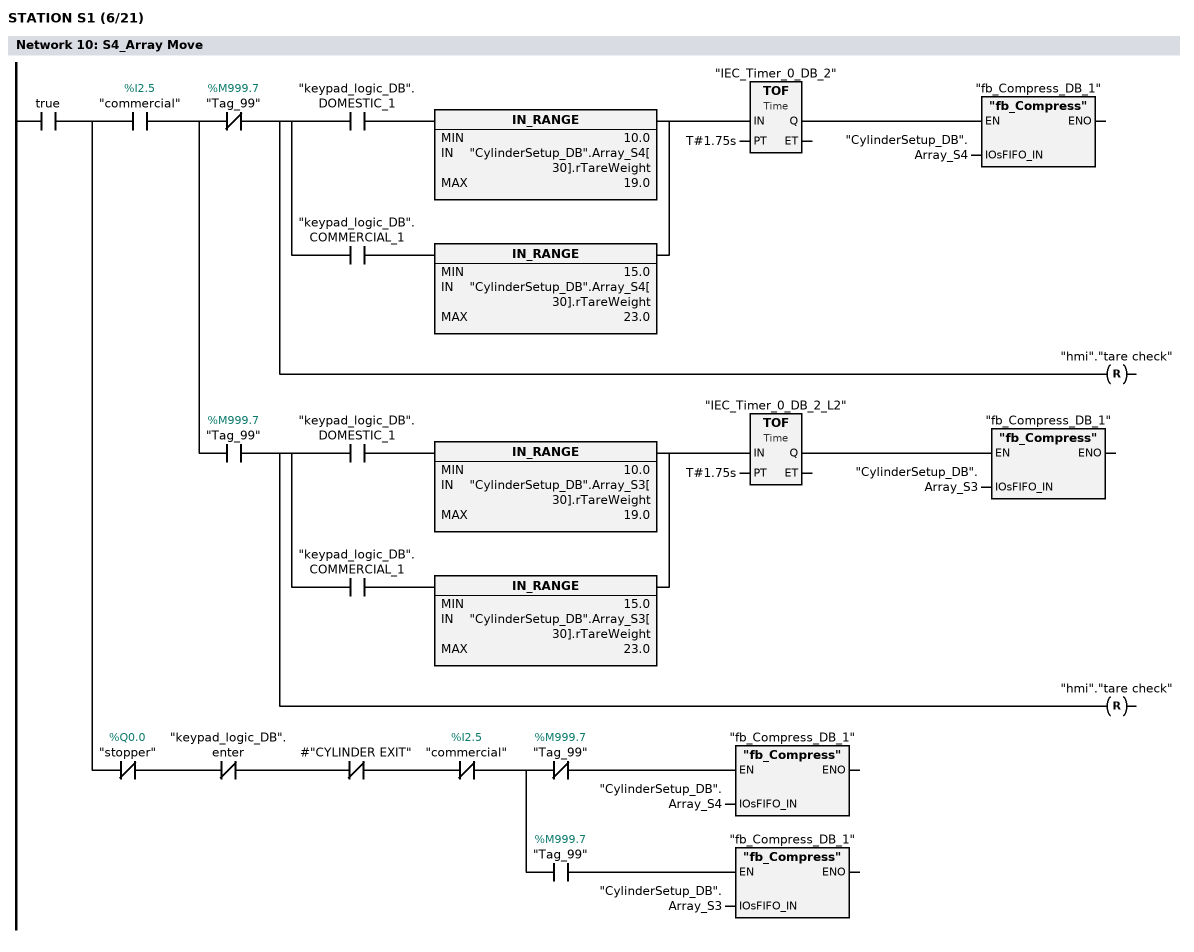
   RUNG wire#powerrail
      Contact( true )
      wire#w1
      Contact( "commercial" )
      wire#w2
      I_Contact( "Tag_99" )
      wire#w3
      Contact( "keypad_logic_DB".DOMESTIC_1 )
      { S7_Templates := "SrcType := Real" } InRange(min := 10.0, in := "CylinderSetup_DB".Array_S4[30].rTareWeight, max := 19.0)
      wire#w4
      { S7_Templates := "time_type := Time" } "IEC_Timer_0_DB_2".TOF(pt := T#1.75s, et =>)
      "fb_Compress_DB_1"(IOsFIFO_IN := "CylinderSetup_DB".Array_S4)
   END_RUNG
   RUNG wire#w3
      Contact( "keypad_logic_DB".COMMERCIAL_1 )
      { S7_Templates := "SrcType := Real" } InRange(min := 15.0, in := "CylinderSetup_DB".Array_S4[30].rTareWeight, max := 23.0)
   END_RUNG wire#w4
   RUNG wire#w3
      R_Coil( "hmi"."tare check" )
   END_RUNG
   RUNG wire#w2
      Contact( "Tag_99" )
      wire#w5
      Contact( "keypad_logic_DB".DOMESTIC_1 )
      { S7_Templates := "SrcType := Real" } InRange(min := 10.0, in := "CylinderSetup_DB".Array_S3[30].rTareWeight, max := 19.0)
      wire#w6
      { S7_Templates := "time_type := Time" } "IEC_Timer_0_DB_2_L2".TOF(pt := T#1.75s, et =>)
      "fb_Compress_DB_1"(IOsFIFO_IN := "CylinderSetup_DB".Array_S3)
   END_RUNG
   RUNG wire#w5
      Contact( "keypad_logic_DB".COMMERCIAL_1 )
      { S7_Templates := "SrcType := Real" } InRange(min := 15.0, in := "CylinderSetup_DB".Array_S3[30].rTareWeight, max := 23.0)
   END_RUNG wire#w6
   RUNG wire#w5
      R_Coil( "hmi"."tare check" )
   END_RUNG
   RUNG wire#w1
      I_Contact( "stopper" )
      I_Contact( "keypad_logic_DB".enter )
      I_Contact( #"CYLINDER EXIT" )
      I_Contact( "commercial" )
      wire#w7
      I_Contact( "Tag_99" )
      "fb_Compress_DB_1"(IOsFIFO_IN := "CylinderSetup_DB".Array_S4)
   END_RUNG
   RUNG wire#w7
      Contact( "Tag_99" )
      "fb_Compress_DB_1"(IOsFIFO_IN := "CylinderSetup_DB".Array_S3)
   END_RUNG
   // the same network as SCL:
   #_w1 := true AND "commercial";
   #_w2 := #_w1 AND NOT "Tag_99";
   "IEC_Timer_0_DB_2".TOF(IN := #_w2 AND (("keypad_logic_DB".DOMESTIC_1 AND (10.0 <= "CylinderSetup_DB".Array_S4[30].rTareWeight) AND ("CylinderSetup_DB".Array_S4[30].rTareWeight <= 19.0)) OR ("keypad_logic_DB".COMMERCIAL_1 AND (15.0 <= "CylinderSetup_DB".Array_S4[30].rTareWeight) AND ("CylinderSetup_DB".Array_S4[30].rTareWeight <= 23.0))),
                          PT := T#1.75s);
   IF "IEC_Timer_0_DB_2".Q THEN
       "fb_Compress_DB_1"(IOsFIFO_IN := "CylinderSetup_DB".Array_S4);   // "fb_Compress"
   END_IF;
   IF #_w2 THEN "hmi"."tare check" := FALSE; END_IF;
   #_w3 := #_w1 AND "Tag_99";
   "IEC_Timer_0_DB_2_L2".TOF(IN := #_w3 AND (("keypad_logic_DB".DOMESTIC_1 AND (10.0 <= "CylinderSetup_DB".Array_S3[30].rTareWeight) AND ("CylinderSetup_DB".Array_S3[30].rTareWeight <= 19.0)) OR ("keypad_logic_DB".COMMERCIAL_1 AND (15.0 <= "CylinderSetup_DB".Array_S3[30].rTareWeight) AND ("CylinderSetup_DB".Array_S3[30].rTareWeight <= 23.0))),
                           PT := T#1.75s);
   IF "IEC_Timer_0_DB_2_L2".Q THEN
       "fb_Compress_DB_1"(IOsFIFO_IN := "CylinderSetup_DB".Array_S3);   // "fb_Compress"
   END_IF;
   IF #_w3 THEN "hmi"."tare check" := FALSE; END_IF;
   #_w4 := true AND NOT "stopper" AND NOT "keypad_logic_DB".enter AND NOT #"CYLINDER EXIT" AND NOT "commercial";
   IF #_w4 AND NOT "Tag_99" THEN
       "fb_Compress_DB_1"(IOsFIFO_IN := "CylinderSetup_DB".Array_S4);   // "fb_Compress"
   END_IF;
   IF #_w4 AND "Tag_99" THEN
       "fb_Compress_DB_1"(IOsFIFO_IN := "CylinderSetup_DB".Array_S3);   // "fb_Compress"
   END_IF;
END_REGION

REGION Network 11: Station1_Rejection NOT USE
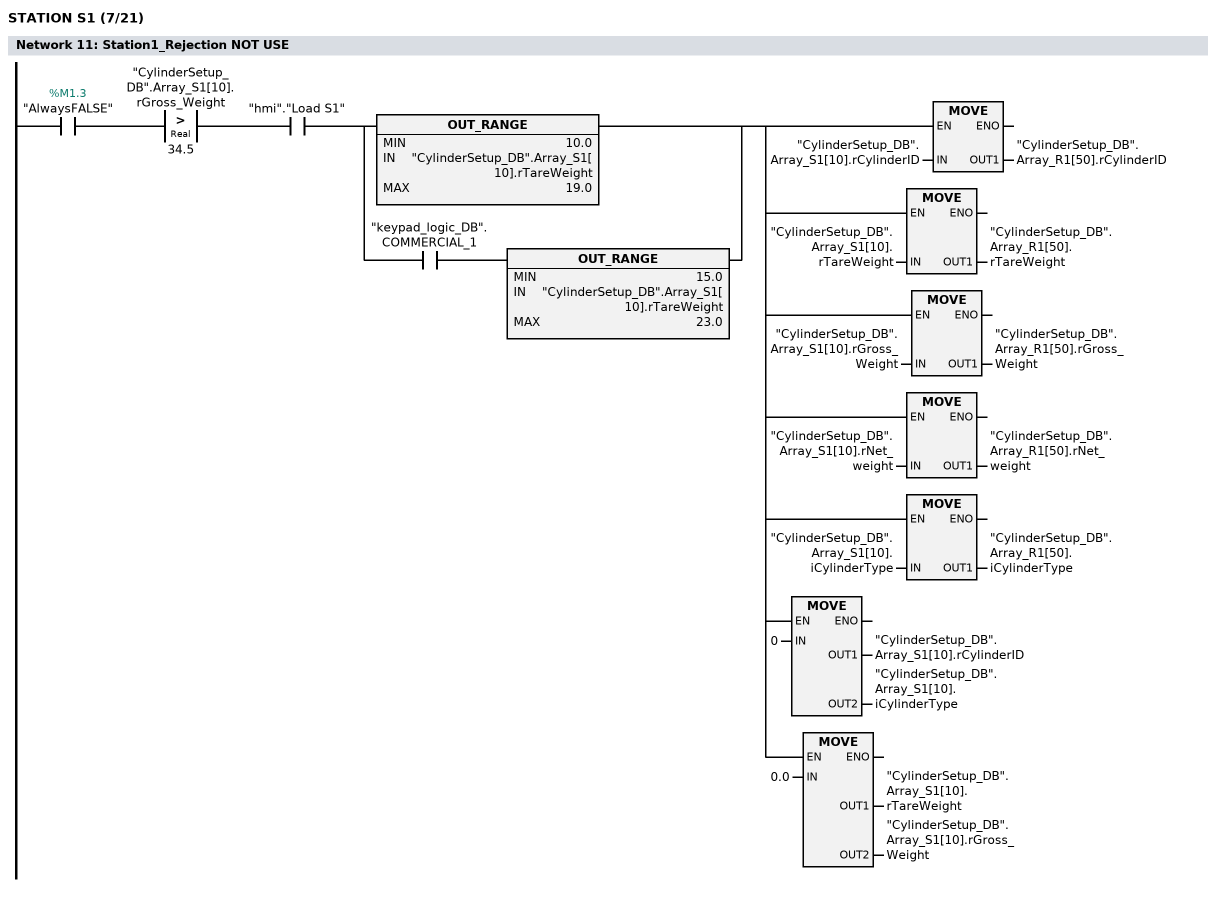
   IF "AlwaysFALSE" AND ("CylinderSetup_DB".Array_S1[10].rGross_Weight > 34.5) AND "hmi"."Load S1" AND (("CylinderSetup_DB".Array_S1[10].rTareWeight < 10.0) OR ("CylinderSetup_DB".Array_S1[10].rTareWeight > 19.0) OR ("keypad_logic_DB".COMMERCIAL_1 AND (("CylinderSetup_DB".Array_S1[10].rTareWeight < 15.0) OR ("CylinderSetup_DB".Array_S1[10].rTareWeight > 23.0)))) THEN
       "CylinderSetup_DB".Array_R1[50].rCylinderID := "CylinderSetup_DB".Array_S1[10].rCylinderID;
       "CylinderSetup_DB".Array_R1[50].rTareWeight := "CylinderSetup_DB".Array_S1[10].rTareWeight;
       "CylinderSetup_DB".Array_R1[50].rGross_Weight := "CylinderSetup_DB".Array_S1[10].rGross_Weight;
       "CylinderSetup_DB".Array_R1[50].rNet_weight := "CylinderSetup_DB".Array_S1[10].rNet_weight;
       "CylinderSetup_DB".Array_R1[50].iCylinderType := "CylinderSetup_DB".Array_S1[10].iCylinderType;
   END_IF;
   #_w1 := "AlwaysFALSE" AND ("CylinderSetup_DB".Array_S1[10].rGross_Weight > 34.5) AND "hmi"."Load S1" AND (("CylinderSetup_DB".Array_S1[10].rTareWeight < 10.0) OR ("CylinderSetup_DB".Array_S1[10].rTareWeight > 19.0) OR ("keypad_logic_DB".COMMERCIAL_1 AND (("CylinderSetup_DB".Array_S1[10].rTareWeight < 15.0) OR ("CylinderSetup_DB".Array_S1[10].rTareWeight > 23.0))));
   IF #_w1 THEN
       "CylinderSetup_DB".Array_S1[10].rCylinderID := 0;
       "CylinderSetup_DB".Array_S1[10].iCylinderType := 0;
       "CylinderSetup_DB".Array_S1[10].rTareWeight := 0.0;
       "CylinderSetup_DB".Array_S1[10].rGross_Weight := 0.0;
   END_IF;
END_REGION

REGION Network 12: data move
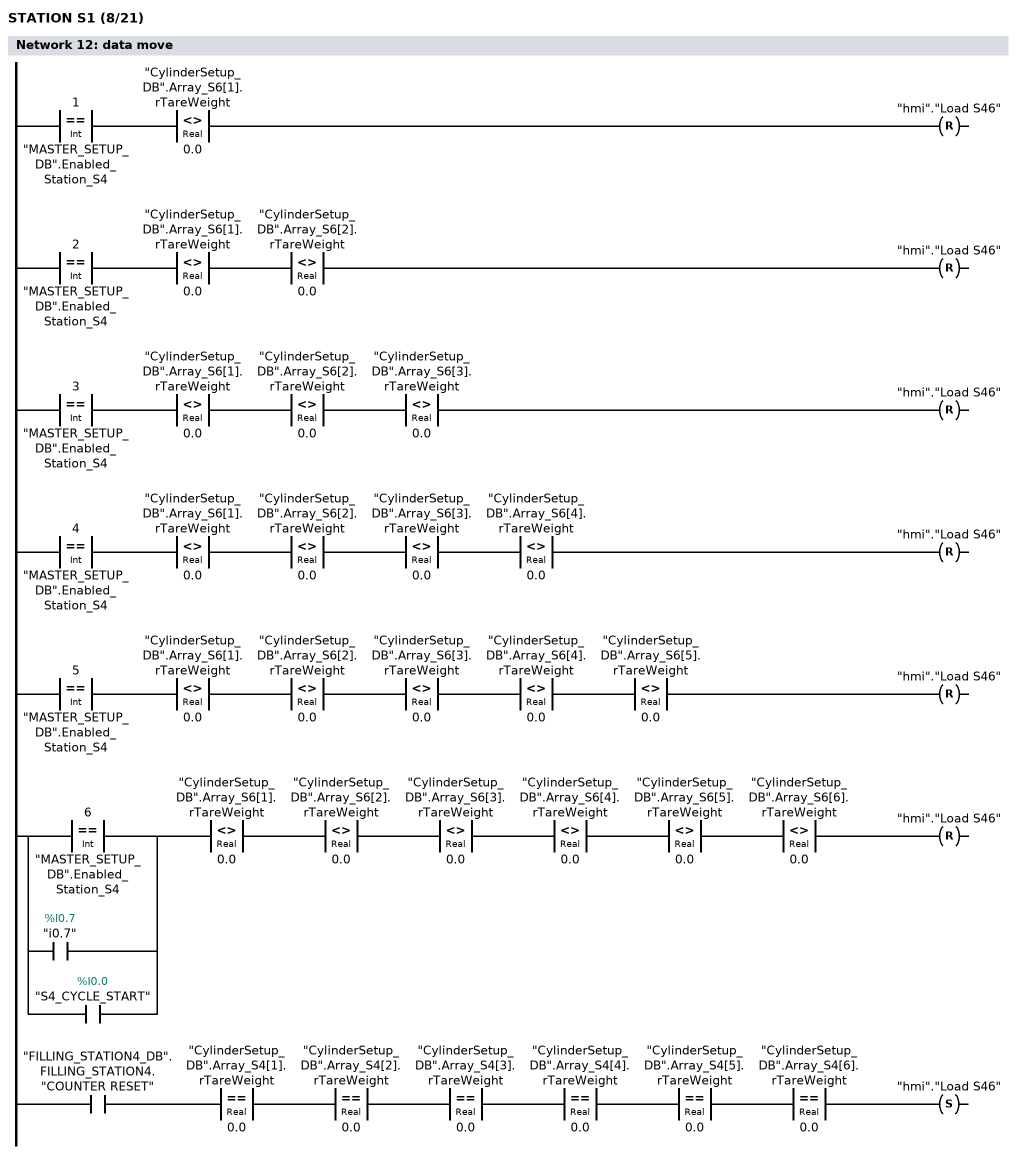
   RUNG wire#powerrail
      { S7_Templates := "SrcType := Int" } EQ_Contact(in1 := 1, in2 := "MASTER_SETUP_DB".Enabled_Station_S4)
      { S7_Templates := "SrcType := Real" } NE_Contact(in1 := "CylinderSetup_DB".Array_S6[1].rTareWeight, in2 := 0.0)
      R_Coil( "hmi"."Load S46" )
   END_RUNG
   RUNG wire#powerrail
      { S7_Templates := "SrcType := Int" } EQ_Contact(in1 := 2, in2 := "MASTER_SETUP_DB".Enabled_Station_S4)
      { S7_Templates := "SrcType := Real" } NE_Contact(in1 := "CylinderSetup_DB".Array_S6[1].rTareWeight, in2 := 0.0)
      { S7_Templates := "SrcType := Real" } NE_Contact(in1 := "CylinderSetup_DB".Array_S6[2].rTareWeight, in2 := 0.0)
      R_Coil( "hmi"."Load S46" )
   END_RUNG
   RUNG wire#powerrail
      { S7_Templates := "SrcType := Int" } EQ_Contact(in1 := 3, in2 := "MASTER_SETUP_DB".Enabled_Station_S4)
      { S7_Templates := "SrcType := Real" } NE_Contact(in1 := "CylinderSetup_DB".Array_S6[1].rTareWeight, in2 := 0.0)
      { S7_Templates := "SrcType := Real" } NE_Contact(in1 := "CylinderSetup_DB".Array_S6[2].rTareWeight, in2 := 0.0)
      { S7_Templates := "SrcType := Real" } NE_Contact(in1 := "CylinderSetup_DB".Array_S6[3].rTareWeight, in2 := 0.0)
      R_Coil( "hmi"."Load S46" )
   END_RUNG
   RUNG wire#powerrail
      { S7_Templates := "SrcType := Int" } EQ_Contact(in1 := 4, in2 := "MASTER_SETUP_DB".Enabled_Station_S4)
      { S7_Templates := "SrcType := Real" } NE_Contact(in1 := "CylinderSetup_DB".Array_S6[1].rTareWeight, in2 := 0.0)
      { S7_Templates := "SrcType := Real" } NE_Contact(in1 := "CylinderSetup_DB".Array_S6[2].rTareWeight, in2 := 0.0)
      { S7_Templates := "SrcType := Real" } NE_Contact(in1 := "CylinderSetup_DB".Array_S6[3].rTareWeight, in2 := 0.0)
      { S7_Templates := "SrcType := Real" } NE_Contact(in1 := "CylinderSetup_DB".Array_S6[4].rTareWeight, in2 := 0.0)
      R_Coil( "hmi"."Load S46" )
   END_RUNG
   RUNG wire#powerrail
      { S7_Templates := "SrcType := Int" } EQ_Contact(in1 := 5, in2 := "MASTER_SETUP_DB".Enabled_Station_S4)
      { S7_Templates := "SrcType := Real" } NE_Contact(in1 := "CylinderSetup_DB".Array_S6[1].rTareWeight, in2 := 0.0)
      { S7_Templates := "SrcType := Real" } NE_Contact(in1 := "CylinderSetup_DB".Array_S6[2].rTareWeight, in2 := 0.0)
      { S7_Templates := "SrcType := Real" } NE_Contact(in1 := "CylinderSetup_DB".Array_S6[3].rTareWeight, in2 := 0.0)
      { S7_Templates := "SrcType := Real" } NE_Contact(in1 := "CylinderSetup_DB".Array_S6[4].rTareWeight, in2 := 0.0)
      { S7_Templates := "SrcType := Real" } NE_Contact(in1 := "CylinderSetup_DB".Array_S6[5].rTareWeight, in2 := 0.0)
      R_Coil( "hmi"."Load S46" )
   END_RUNG
   RUNG wire#powerrail
      { S7_Templates := "SrcType := Int" } EQ_Contact(in1 := 6, in2 := "MASTER_SETUP_DB".Enabled_Station_S4)
      wire#w1
      { S7_Templates := "SrcType := Real" } NE_Contact(in1 := "CylinderSetup_DB".Array_S6[1].rTareWeight, in2 := 0.0)
      { S7_Templates := "SrcType := Real" } NE_Contact(in1 := "CylinderSetup_DB".Array_S6[2].rTareWeight, in2 := 0.0)
      { S7_Templates := "SrcType := Real" } NE_Contact(in1 := "CylinderSetup_DB".Array_S6[3].rTareWeight, in2 := 0.0)
      { S7_Templates := "SrcType := Real" } NE_Contact(in1 := "CylinderSetup_DB".Array_S6[4].rTareWeight, in2 := 0.0)
      { S7_Templates := "SrcType := Real" } NE_Contact(in1 := "CylinderSetup_DB".Array_S6[5].rTareWeight, in2 := 0.0)
      { S7_Templates := "SrcType := Real" } NE_Contact(in1 := "CylinderSetup_DB".Array_S6[6].rTareWeight, in2 := 0.0)
      R_Coil( "hmi"."Load S46" )
   END_RUNG
   RUNG wire#powerrail
      Contact( "i0.7" )
   END_RUNG wire#w1
   RUNG wire#powerrail
      Contact( "S4_CYCLE_START" )
   END_RUNG wire#w1
   RUNG wire#powerrail
      Contact( "FILLING_STATION4_DB".FILLING_STATION4."COUNTER RESET" )
      { S7_Templates := "SrcType := Real" } EQ_Contact(in1 := "CylinderSetup_DB".Array_S4[1].rTareWeight, in2 := 0.0)
      { S7_Templates := "SrcType := Real" } EQ_Contact(in1 := "CylinderSetup_DB".Array_S4[2].rTareWeight, in2 := 0.0)
      { S7_Templates := "SrcType := Real" } EQ_Contact(in1 := "CylinderSetup_DB".Array_S4[3].rTareWeight, in2 := 0.0)
      { S7_Templates := "SrcType := Real" } EQ_Contact(in1 := "CylinderSetup_DB".Array_S4[4].rTareWeight, in2 := 0.0)
      { S7_Templates := "SrcType := Real" } EQ_Contact(in1 := "CylinderSetup_DB".Array_S4[5].rTareWeight, in2 := 0.0)
      { S7_Templates := "SrcType := Real" } EQ_Contact(in1 := "CylinderSetup_DB".Array_S4[6].rTareWeight, in2 := 0.0)
      S_Coil( "hmi"."Load S46" )
   END_RUNG
   // the same network as SCL:
   IF (1 = "MASTER_SETUP_DB".Enabled_Station_S4) AND ("CylinderSetup_DB".Array_S6[1].rTareWeight <> 0.0) THEN
       "hmi"."Load S46" := FALSE;
   END_IF;
   IF (2 = "MASTER_SETUP_DB".Enabled_Station_S4) AND ("CylinderSetup_DB".Array_S6[1].rTareWeight <> 0.0) AND ("CylinderSetup_DB".Array_S6[2].rTareWeight <> 0.0) THEN
       "hmi"."Load S46" := FALSE;
   END_IF;
   IF (3 = "MASTER_SETUP_DB".Enabled_Station_S4) AND ("CylinderSetup_DB".Array_S6[1].rTareWeight <> 0.0) AND ("CylinderSetup_DB".Array_S6[2].rTareWeight <> 0.0) AND ("CylinderSetup_DB".Array_S6[3].rTareWeight <> 0.0) THEN
       "hmi"."Load S46" := FALSE;
   END_IF;
   IF (4 = "MASTER_SETUP_DB".Enabled_Station_S4) AND ("CylinderSetup_DB".Array_S6[1].rTareWeight <> 0.0) AND ("CylinderSetup_DB".Array_S6[2].rTareWeight <> 0.0) AND ("CylinderSetup_DB".Array_S6[3].rTareWeight <> 0.0) AND ("CylinderSetup_DB".Array_S6[4].rTareWeight <> 0.0) THEN
       "hmi"."Load S46" := FALSE;
   END_IF;
   IF (5 = "MASTER_SETUP_DB".Enabled_Station_S4) AND ("CylinderSetup_DB".Array_S6[1].rTareWeight <> 0.0) AND ("CylinderSetup_DB".Array_S6[2].rTareWeight <> 0.0) AND ("CylinderSetup_DB".Array_S6[3].rTareWeight <> 0.0) AND ("CylinderSetup_DB".Array_S6[4].rTareWeight <> 0.0) AND ("CylinderSetup_DB".Array_S6[5].rTareWeight <> 0.0) THEN
       "hmi"."Load S46" := FALSE;
   END_IF;
   IF ((6 = "MASTER_SETUP_DB".Enabled_Station_S4) OR "i0.7" OR "S4_CYCLE_START") AND ("CylinderSetup_DB".Array_S6[1].rTareWeight <> 0.0) AND ("CylinderSetup_DB".Array_S6[2].rTareWeight <> 0.0) AND ("CylinderSetup_DB".Array_S6[3].rTareWeight <> 0.0) AND ("CylinderSetup_DB".Array_S6[4].rTareWeight <> 0.0) AND ("CylinderSetup_DB".Array_S6[5].rTareWeight <> 0.0) AND ("CylinderSetup_DB".Array_S6[6].rTareWeight <> 0.0) THEN
       "hmi"."Load S46" := FALSE;
   END_IF;
   IF "FILLING_STATION4_DB".FILLING_STATION4."COUNTER RESET" AND ("CylinderSetup_DB".Array_S4[1].rTareWeight = 0.0) AND ("CylinderSetup_DB".Array_S4[2].rTareWeight = 0.0) AND ("CylinderSetup_DB".Array_S4[3].rTareWeight = 0.0) AND ("CylinderSetup_DB".Array_S4[4].rTareWeight = 0.0) AND ("CylinderSetup_DB".Array_S4[5].rTareWeight = 0.0) AND ("CylinderSetup_DB".Array_S4[6].rTareWeight = 0.0) THEN
       "hmi"."Load S46" := TRUE;
   END_IF;
END_REGION

REGION Network 13: S6_TO_S8 SAME L1 exit
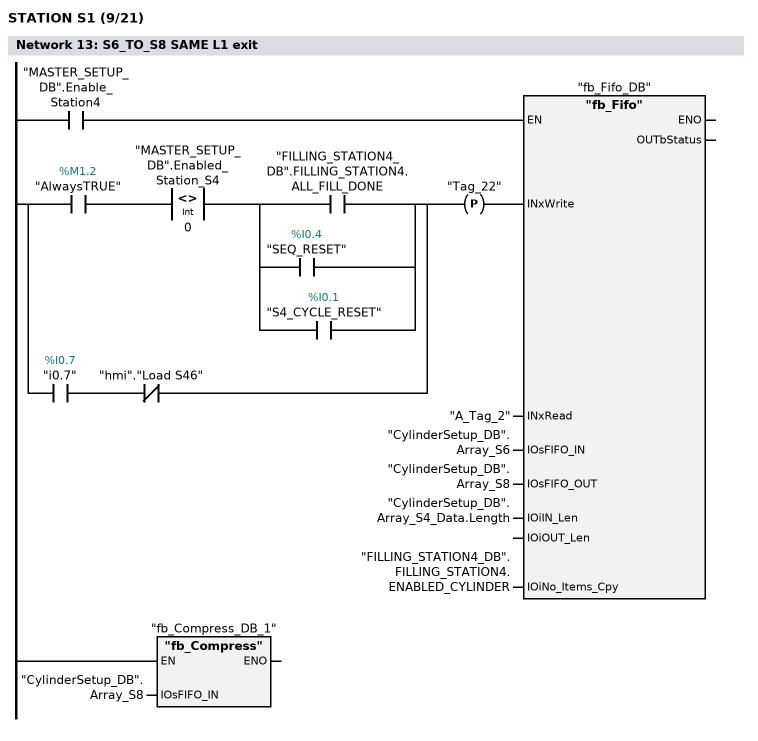
   RUNG wire#powerrail
      Contact( "MASTER_SETUP_DB".Enable_Station4 )
      "fb_Fifo_DB"(INxWrite := wire#w3, INxRead := "A_Tag_2", IOsFIFO_IN := "CylinderSetup_DB".Array_S6, IOsFIFO_OUT := "CylinderSetup_DB".Array_S8, IOiIN_Len := "CylinderSetup_DB".Array_S4_Data.Length, IOiOUT_Len :=, IOiNo_Items_Cpy := "FILLING_STATION4_DB".FILLING_STATION4.ENABLED_CYLINDER, OUTbStatus =>)
   END_RUNG
   RUNG wire#powerrail
      Contact( "AlwaysTRUE" )
      { S7_Templates := "SrcType := Int" } NE_Contact(in1 := "MASTER_SETUP_DB".Enabled_Station_S4, in2 := 0)
      wire#w1
      Contact( "FILLING_STATION4_DB".FILLING_STATION4.ALL_FILL_DONE )
      wire#w2
      P_Trig( "Tag_22" )
   END_RUNG wire#w3
   RUNG wire#w1
      Contact( "SEQ_RESET" )
   END_RUNG wire#w2
   RUNG wire#w1
      Contact( "S4_CYCLE_RESET" )
   END_RUNG wire#w2
   RUNG wire#powerrail
      Contact( "i0.7" )
      I_Contact( "hmi"."Load S46" )
   END_RUNG wire#w2
   RUNG wire#powerrail
      "fb_Compress_DB_1"(IOsFIFO_IN := "CylinderSetup_DB".Array_S8)
   END_RUNG
   // the same network as SCL:
   #_w1 := ("AlwaysTRUE" AND ("MASTER_SETUP_DB".Enabled_Station_S4 <> 0) AND ("FILLING_STATION4_DB".FILLING_STATION4.ALL_FILL_DONE OR "SEQ_RESET" OR "S4_CYCLE_RESET")) OR ("i0.7" AND NOT "hmi"."Load S46");
   #_w2 := #_w1 AND NOT "Tag_22";   // rising edge
   "Tag_22" := #_w1;
   IF "MASTER_SETUP_DB".Enable_Station4 THEN
       "fb_Fifo_DB"(INxWrite := #_w2,   // "fb_Fifo"
                    INxRead := "A_Tag_2",
                    IOsFIFO_IN := "CylinderSetup_DB".Array_S6,
                    IOsFIFO_OUT := "CylinderSetup_DB".Array_S8,
                    IOiIN_Len := "CylinderSetup_DB".Array_S4_Data.Length,
                    IOiNo_Items_Cpy := "FILLING_STATION4_DB".FILLING_STATION4.ENABLED_CYLINDER);
   END_IF;
   "fb_Compress_DB_1"(IOsFIFO_IN := "CylinderSetup_DB".Array_S8);   // "fb_Compress"
END_REGION

